(* PLC project Neotec skyrailer, Hydac System GmbH CoDeSys CoDeSys V3.x *)
(* stored: companyURL http://www.hydac.com/, contentDescription This content was automatically generated. Please do not edit., creationDateTime 2025-04-18T16:40:50.760, modificationDateTime 2025-04-18T16:40:50.760 *)

TYPE EBRAKETESTSELECTED : (GE_OSCI_SERVICE_BRAKE := 0, GE_FIXE_SERVICE_BRAKE := 1, GE_OSCI_PARKING_BRAKE := 2, GE_FIXE_PARKING_BRAKE := 3, GE_SERVICE_BRAKES := 4, GE_PARKING_BRAKES := 5, GE_NO_BRAKE := 6, GE_FIXE_2ND_PARKING_BRAKE := 7, GE_OSCI_2ND_PARKING_BRAKE := 8);
END_TYPE

TYPE ECONTROLPOST : (GE_POST_NO_POST := 0, GE_POST_RADIO := 1, GE_POST_NACELLE := 2, GE_POST_TURRET := 3);
END_TYPE

TYPE ECOUNTRY : (GE_FRANCE := 0, GE_SWITZERLAND := 1, GE_UNITED_KINGDOM := 2, GE_AUSTRALIA := 3);
END_TYPE

TYPE EDIGSTATUS : (GE_DIG_OFF := 0, GE_DIG_ON := 1, GE_DIG_ERROR := 2, GE_DIG_UNDEF := 3);
END_TYPE

TYPE EDISTATE : (GE_DI_OFF := 0, GE_DI_ON := 1, GE_DI_ERROR := 2, GE_DI_UNDEF := 3);
END_TYPE

TYPE EERRORSTATUS48XS : (GE_IO_E_OK := 0, GE_IO_E_BUSY := 2, GE_IO_E_UNKNOWN := 3, GE_IO_E_CHANNEL_BUSY := 32, GE_IO_E_CHANNEL_NOT_CONFIGURED := 33, GE_IO_E_FET_PROTECTION := 35, GE_IO_E_ADC_NOT_FINISH := 90, GE_IO_E_PWD_CAPTURE_ERROR := 100, GE_IO_E_PWD_NOT_FINISHED := 101, GE_IO_E_PWD_OPEN_LOAD := 102, GE_IO_E_PWD_SHORT_CIRCUIT := 103, GE_IO_E_PWD_TIMER_OVERFLOW := 104, GE_IO_E_PWD_HIGH_LEVEL := 105, GE_IO_E_PWD_LOW_LEVEL := 106, GE_IO_E_PWD_CURRENT_THRESHOLD_HIGH := 107, GE_IO_E_PWD_CURRENT_THRESHOLD_LOW := 108, GE_IO_E_DO_OPEN_LOAD := 110, GE_IO_E_DO_SHORT_CIRCUIT := 111, GE_IO_E_DO_DIAG_NOT_FINISHED := 112);
END_TYPE

TYPE EMANIPULATORPOSITION : (GE_NEUTRAL := 0, GE_AV := 1, GE_AR := 2, GE_ERROR := 3);
END_TYPE

TYPE EMOTORSTATE : (GE_Stopped := 0, GE_PreStart := 1, GE_Starting := 2, GE_WarmUp := 3, GE_Running := 4, GE_CoolDown := 5, GE_Stopping := 6, GE_PostRun := 7);
END_TYPE

TYPE EMOVENACELLEMODE : (GE_NO_MODE := 0, GE_OFFRAIL_RADIOCONTOL_MODE := 1, GE_RAIL_NACELLE_MODE := 2, GE_TURRET_MODE := 3);
END_TYPE

TYPE EOFFRAILMODE : (GE_NO_OFFRAIL_MODE := 0, GE_TRANSPORT_OFFRAIL_MODE := 1, GE_WORK_OFFRAIL_MODE := 2, GE_WORSHOP_OFFRAIL_MODE := 3);
END_TYPE

TYPE EPOSJOY : (GE_AV_JOY := 0, GE_NEU_JOY := 1, GE_AR_JOY := 2);
END_TYPE

TYPE EPROSTATUS : (GE_PRO_OFF := 0, GE_PRO_ON := 1, GE_PRO_ERROR := 2, GE_PRO_NOT_INSTALLED := 3, GE_PRO_NO_DUTY_CYCLE := 4, GE_PRO_MIN_DUTY_CYCLE := 5);
END_TYPE

TYPE ERAILSPEEDMODE : (GE_NO_SPEED_MAX_RAIL_MODE := 0, GE_ACCESS_SITE_MODE := 1, GE_HIGH_SPEED := 2, GE_LOW_SPEED := 3, GE_LOW_SPEED_BRAKE_TEST_NEEDED := 4, GE_BRAKE_TEST_SPEED_RUNNING := 5, GE_BREAK_IN_BRAKE_SPEED_RUNNING := 6);
END_TYPE

TYPE ERAILTRANSLATIONDIRECTION : (GE_AV_RAIL_DIR := 0, GE_AR_RAIL_DIR := 1, GE_STOP_RAIL_DIR := 2);
END_TYPE

TYPE ERAILWORKMODE : (GE_NO_RAIL_WORK_MODE := 0, GE_BILATERAL_MODE := 1, GE_ALO_MODE := 2, GE_MULTILANE_MODE := 3);
END_TYPE

TYPE ESTATEBOOL2BITS : (GE_OFF := 0, GE_ON := 1, GE_ERR := 2, GE_NA := 3);
END_TYPE

TYPE ESTATEHEARTBEAT : (GE_BOOT_UP := 0, GE_STOPPED := 4, GE_OPERATIONAL := 5, GE_PRE_OPERATIONAL := 127);
END_TYPE

TYPE ESTATESERVICEBRAKERAIL : (GE_DEFINE_BRAKE := 0, GE_AV_SERVICE_BRAKE := 1, GE_AR_SERVICE_BRAKE := 2);
END_TYPE

TYPE ETRANSPORTPOSITION : (GE_NO_TRANSPORT_POSITION := 0, GE_OFFRAIL_TRANSPORT_POSITION := 1, GE_RAIL_TRANSPORT_POSITION := 2);
END_TYPE

TYPE EWDSTATE : (GE_RUNNING := 6, GE_TRIGGERED := 9);
END_TYPE

VAR_GLOBAL CONSTANT  (* GlobalConsts *)
  J1939_SA_DISPLAY : BYTE := 16#2f;  (* Display *)
END_VAR

VAR_GLOBAL  (* GCanMessages *)
  g_CanMessages_Msg8C1SendToOpus : Msg8C1SendToOpusMessageClass;
  g_CanMessages_Msg9C1SendToOpus : Msg9C1SendToOpusMessageClass;
  g_CanMessages_Msg1C0SendToEvision7 : Msg1C0SendToEvision7MessageClass;
  g_CanMessages_Msg2C0SendToEvision7 : Msg2C0SendToEvision7MessageClass;
  g_CanMessages_Msg3C0SendToEvision7 : Msg3C0SendToEvision7MessageClass;
  g_CanMessages_Msg4C0SendToEvision7 : Msg4C0SendToEvision7MessageClass;
  g_CanMessages_Msg5C0SendToEvision7 : Msg5C0SendToEvision7MessageClass;
  g_CanMessages_Msg6C0SendToEvision7 : Msg6C0SendToEvision7MessageClass;
  g_CanMessages_Msg7C0SendToEvision7 : Msg7C0SendToEvision7MessageClass;
  g_CanMessages_Msg8C0SendToEvision7 : Msg8C0SendToEvision7MessageClass;
  g_CanMessages_Msg9C0SendToEvision7 : Msg9C0SendToEvision7MessageClass;
  g_CanMessages_Msg10C0SendToEvision7 : Msg10C0SendToEvision7MessageClass;
  g_CanMessages_Msg11C0SendToEvision7 : Msg11C0SendToEvision7MessageClass;
  g_CanMessages_Msg12C0SendToEvision7 : Msg12C0SendToEvision7MessageClass;
  g_CanMessages_Msg13C0SendToEvision7 : Msg13C0SendToEvision7MessageClass;
  g_CanMessages_Msg14C0SendToEvision7 : Msg14C0SendToEvision7MessageClass;
  g_CanMessages_Msg15C0SendToEvision7 : Msg15C0SendToEvision7MessageClass;
  g_CanMessages_MsgDebugC0SendToEvision7 : MsgDebugC0SendToEvision7MessageClass;
  g_CanMessages_Msg1C1SendToEvision7 : Msg1C1SendToEvision7MessageClass;
  g_CanMessages_Msg2C1SendToEvision7 : Msg2C1SendToEvision7MessageClass;
  g_CanMessages_Msg3C1SendToEvision7 : Msg3C1SendToEvision7MessageClass;
  g_CanMessages_Msg4C1SendToEvision7 : Msg4C1SendToEvision7MessageClass;
  g_CanMessages_Msg5C1SendToEvision7 : Msg5C1SendToEvision7MessageClass;
  g_CanMessages_Msg6C1SendToEvision7 : Msg6C1SendToEvision7MessageClass;
  g_CanMessages_Msg7C1SendToEvision7 : Msg7C1SendToEvision7MessageClass;
  g_CanMessages_Msg8C1SendToEvision7 : Msg8C1SendToEvision7MessageClass;
  g_CanMessages_Msg9C1SendToEvision7 : Msg9C1SendToEvision7MessageClass;
  g_CanMessages_Msg10C1SendToEvision7 : Msg10C1SendToEvision7MessageClass;
  g_CanMessages_Msg11C1SendToEvision7 : Msg11C1SendToEvision7MessageClass;
  g_CanMessages_Msg12C1SendToEvision7 : Msg12C1SendToEvision7MessageClass;
  g_CanMessages_Msg13C1SendToEvision7 : Msg13C1SendToEvision7MessageClass;
  g_CanMessages_Msg14C1SendToEvision7 : Msg14C1SendToEvision7MessageClass;
  g_CanMessages_MsgDebugC1SendToEvision7 : MsgDebugC1SendToEvision7MessageClass;
  g_CanMessages_Msg1RcvFromEvision7 : Msg1RcvFromEvision7MessageClass;
END_VAR

VAR_GLOBAL CONSTANT  (* GeneratedCanConsts *)
  CID_MSG8C1SENDTOOPUS : DWORD := 16#506;
  CID_MSG9C1SENDTOOPUS : DWORD := 16#606;
  CID_MSG1C0SENDTOEVISION7 : DWORD := 16#C0D701;
  CID_MSG2C0SENDTOEVISION7 : DWORD := 16#C0D702;
  CID_MSG3C0SENDTOEVISION7 : DWORD := 16#C0D703;
  CID_MSG4C0SENDTOEVISION7 : DWORD := 16#C0D704;
  CID_MSG5C0SENDTOEVISION7 : DWORD := 16#C0D705;
  CID_MSG6C0SENDTOEVISION7 : DWORD := 16#C0D706;
  CID_MSG7C0SENDTOEVISION7 : DWORD := 16#C0D707;
  CID_MSG8C0SENDTOEVISION7 : DWORD := 16#C0D708;
  CID_MSG9C0SENDTOEVISION7 : DWORD := 16#C0D709;
  CID_MSG10C0SENDTOEVISION7 : DWORD := 16#C0D70A;
  CID_MSG11C0SENDTOEVISION7 : DWORD := 16#C0D70B;
  CID_MSG12C0SENDTOEVISION7 : DWORD := 16#C0D70C;
  CID_MSG13C0SENDTOEVISION7 : DWORD := 16#C0D70D;
  CID_MSG14C0SENDTOEVISION7 : DWORD := 16#C0D70E;
  CID_MSG15C0SENDTOEVISION7 : DWORD := 16#C0D70F;
  CID_MSGDEBUGC0SENDTOEVISION7 : DWORD := 16#C0D711;
  CID_MSG1C1SENDTOEVISION7 : DWORD := 16#C1D701;
  CID_MSG2C1SENDTOEVISION7 : DWORD := 16#C1D702;
  CID_MSG3C1SENDTOEVISION7 : DWORD := 16#C1D703;
  CID_MSG4C1SENDTOEVISION7 : DWORD := 16#C1D704;
  CID_MSG5C1SENDTOEVISION7 : DWORD := 16#C1D705;
  CID_MSG6C1SENDTOEVISION7 : DWORD := 16#C1D706;
  CID_MSG7C1SENDTOEVISION7 : DWORD := 16#C1D707;
  CID_MSG8C1SENDTOEVISION7 : DWORD := 16#C1D708;
  CID_MSG9C1SENDTOEVISION7 : DWORD := 16#C1D709;
  CID_MSG10C1SENDTOEVISION7 : DWORD := 16#C1D70A;
  CID_MSG11C1SENDTOEVISION7 : DWORD := 16#C1D70B;
  CID_MSG12C1SENDTOEVISION7 : DWORD := 16#C1D70C;
  CID_MSG13C1SENDTOEVISION7 : DWORD := 16#C1D70D;
  CID_MSG14C1SENDTOEVISION7 : DWORD := 16#C1D70E;
  CID_MSGDEBUGC1SENDTOEVISION7 : DWORD := 16#C1D712;
  CID_MSG1RCVFROMEVISION7 : DWORD := 16#D7CF01;
END_VAR

VAR_GLOBAL CONSTANT  (* GConsts *)
  J1939_SA_C0 : BYTE := 16#20;
  J1939_SA_C1 : BYTE := 16#21;
  J1939_SA_C2 : BYTE := 16#2F;
  CID_P2P_C0 : DWORD := 16#18EE0020;
  CID_P2P_C1 : DWORD := 16#18EE0021;
END_VAR

FUNCTION_BLOCK CanDispatcherClass IMPLEMENTS ICanDispatcher
  VAR
    fMessage : VBasic.CanMessageClass;
    cycleTimerHst : IntervalTimerClass;  (* Determines how much time lays between the sending of HST can messages (CAN 0) *)
    can0 : VBasic.CanManagerClass;  (* CAN 0: C0_C1_CAN_0 *)
    j1939_can0 : J1939ReceiverClass;
    can1 : VBasic.CanManagerClass;  (* CAN 1: CO_C1_CAN_1_TTC48XS *)
    j1939_can1 : J1939ReceiverClass;
  END_VAR
  VAR_INPUT
    Can0MessagesSent : BoolCanSignalClass;
    Can1MessagesSent : BoolCanSignalClass;
  END_VAR

            
          

METHOD Initialize
                  // **********************************************************************************************************************
// *  AUTO-GENERATED:  PdtCodeBuilder.dll (Version: 1.2.7, Build: 080)
// *  Itf-Version:     1.7.0
// *  Pdt-Version:     2.11.72.172
// *  Pdt-ProjVersion: 0.0.0
// *  Match-Version:   07.04.00.00
// *  Copyright (C) 2012 HYDAC SYSTEM GMBH -  All rights reserved.
// *  Entwicklungsbüro Berlin - Zum Kiesberg 16 - D-14979 Großbeeren
// *  2025-04-18 16:40:50 created
// **********************************************************************************************************************

// Initialize the can bus objects

can0.NetId := 0;
can0.Baudrate := eCanBaudrate.BAUDRATE_250_KBITS;
can0.Initialize();

g_CanMessages_Msg1C0SendToEvision7.Initialize(ADR(can0), CID_MSG1C0SENDTOEVISION7, TCanMessageType.RX, 1000(*Timeout*), 0(*Spn*), 255(*Fmi*), 255(*FmiExt*), eErrorType.ERROR(*ErrType*), eErrorSeverity.CAT0_NO(*ErrCat*), eCanIdFormat.EXTENDED);
g_CanMessages_Msg2C0SendToEvision7.Initialize(ADR(can0), CID_MSG2C0SENDTOEVISION7, TCanMessageType.RX, 1000(*Timeout*), 0(*Spn*), 255(*Fmi*), 255(*FmiExt*), eErrorType.ERROR(*ErrType*), eErrorSeverity.CAT0_NO(*ErrCat*), eCanIdFormat.EXTENDED);
g_CanMessages_Msg3C0SendToEvision7.Initialize(ADR(can0), CID_MSG3C0SENDTOEVISION7, TCanMessageType.RX, 1000(*Timeout*), 0(*Spn*), 255(*Fmi*), 255(*FmiExt*), eErrorType.ERROR(*ErrType*), eErrorSeverity.CAT0_NO(*ErrCat*), eCanIdFormat.EXTENDED);
g_CanMessages_Msg4C0SendToEvision7.Initialize(ADR(can0), CID_MSG4C0SENDTOEVISION7, TCanMessageType.RX, 1000(*Timeout*), 0(*Spn*), 255(*Fmi*), 255(*FmiExt*), eErrorType.ERROR(*ErrType*), eErrorSeverity.CAT0_NO(*ErrCat*), eCanIdFormat.EXTENDED);
g_CanMessages_Msg5C0SendToEvision7.Initialize(ADR(can0), CID_MSG5C0SENDTOEVISION7, TCanMessageType.RX, 1000(*Timeout*), 0(*Spn*), 255(*Fmi*), 255(*FmiExt*), eErrorType.ERROR(*ErrType*), eErrorSeverity.CAT0_NO(*ErrCat*), eCanIdFormat.EXTENDED);
g_CanMessages_Msg6C0SendToEvision7.Initialize(ADR(can0), CID_MSG6C0SENDTOEVISION7, TCanMessageType.RX, 1000(*Timeout*), 0(*Spn*), 255(*Fmi*), 255(*FmiExt*), eErrorType.ERROR(*ErrType*), eErrorSeverity.CAT0_NO(*ErrCat*), eCanIdFormat.EXTENDED);
g_CanMessages_Msg7C0SendToEvision7.Initialize(ADR(can0), CID_MSG7C0SENDTOEVISION7, TCanMessageType.RX, 1000(*Timeout*), 0(*Spn*), 255(*Fmi*), 255(*FmiExt*), eErrorType.ERROR(*ErrType*), eErrorSeverity.CAT0_NO(*ErrCat*), eCanIdFormat.EXTENDED);
g_CanMessages_Msg8C0SendToEvision7.Initialize(ADR(can0), CID_MSG8C0SENDTOEVISION7, TCanMessageType.RX, 1000(*Timeout*), 0(*Spn*), 255(*Fmi*), 255(*FmiExt*), eErrorType.ERROR(*ErrType*), eErrorSeverity.CAT0_NO(*ErrCat*), eCanIdFormat.EXTENDED);
g_CanMessages_Msg9C0SendToEvision7.Initialize(ADR(can0), CID_MSG9C0SENDTOEVISION7, TCanMessageType.RX, 1000(*Timeout*), 0(*Spn*), 255(*Fmi*), 255(*FmiExt*), eErrorType.ERROR(*ErrType*), eErrorSeverity.CAT0_NO(*ErrCat*), eCanIdFormat.EXTENDED);
g_CanMessages_Msg10C0SendToEvision7.Initialize(ADR(can0), CID_MSG10C0SENDTOEVISION7, TCanMessageType.RX, 1000(*Timeout*), 0(*Spn*), 255(*Fmi*), 255(*FmiExt*), eErrorType.ERROR(*ErrType*), eErrorSeverity.CAT0_NO(*ErrCat*), eCanIdFormat.EXTENDED);
g_CanMessages_Msg11C0SendToEvision7.Initialize(ADR(can0), CID_MSG11C0SENDTOEVISION7, TCanMessageType.RX, 1000(*Timeout*), 0(*Spn*), 255(*Fmi*), 255(*FmiExt*), eErrorType.ERROR(*ErrType*), eErrorSeverity.CAT0_NO(*ErrCat*), eCanIdFormat.EXTENDED);
g_CanMessages_Msg12C0SendToEvision7.Initialize(ADR(can0), CID_MSG12C0SENDTOEVISION7, TCanMessageType.RX, 1000(*Timeout*), 0(*Spn*), 255(*Fmi*), 255(*FmiExt*), eErrorType.ERROR(*ErrType*), eErrorSeverity.CAT0_NO(*ErrCat*), eCanIdFormat.EXTENDED);
g_CanMessages_Msg13C0SendToEvision7.Initialize(ADR(can0), CID_MSG13C0SENDTOEVISION7, TCanMessageType.RX, 1000(*Timeout*), 0(*Spn*), 255(*Fmi*), 255(*FmiExt*), eErrorType.ERROR(*ErrType*), eErrorSeverity.CAT0_NO(*ErrCat*), eCanIdFormat.EXTENDED);
g_CanMessages_Msg14C0SendToEvision7.Initialize(ADR(can0), CID_MSG14C0SENDTOEVISION7, TCanMessageType.RX, 1000(*Timeout*), 1544(*Spn*), 31(*Fmi*), 255(*FmiExt*), eErrorType.ERROR(*ErrType*), eErrorSeverity.CAT0_NO(*ErrCat*), eCanIdFormat.EXTENDED);
g_CanMessages_Msg15C0SendToEvision7.Initialize(ADR(can0), CID_MSG15C0SENDTOEVISION7, TCanMessageType.RX, 1000(*Timeout*), 1555(*Spn*), 31(*Fmi*), 255(*FmiExt*), eErrorType.ERROR(*ErrType*), eErrorSeverity.CAT0_NO(*ErrCat*), eCanIdFormat.EXTENDED);
g_CanMessages_MsgDebugC0SendToEvision7.Initialize(ADR(can0), CID_MSGDEBUGC0SENDTOEVISION7, TCanMessageType.RX, 1000(*Timeout*), 0(*Spn*), 255(*Fmi*), 255(*FmiExt*), eErrorType.ERROR(*ErrType*), eErrorSeverity.CAT0_NO(*ErrCat*), eCanIdFormat.EXTENDED);
g_CanMessages_Msg1C1SendToEvision7.Initialize(ADR(can0), CID_MSG1C1SENDTOEVISION7, TCanMessageType.RX, 1000(*Timeout*), 0(*Spn*), 255(*Fmi*), 255(*FmiExt*), eErrorType.ERROR(*ErrType*), eErrorSeverity.CAT0_NO(*ErrCat*), eCanIdFormat.EXTENDED);
g_CanMessages_Msg2C1SendToEvision7.Initialize(ADR(can0), CID_MSG2C1SENDTOEVISION7, TCanMessageType.RX, 1000(*Timeout*), 0(*Spn*), 255(*Fmi*), 255(*FmiExt*), eErrorType.ERROR(*ErrType*), eErrorSeverity.CAT0_NO(*ErrCat*), eCanIdFormat.EXTENDED);
g_CanMessages_Msg3C1SendToEvision7.Initialize(ADR(can0), CID_MSG3C1SENDTOEVISION7, TCanMessageType.RX, 1000(*Timeout*), 0(*Spn*), 255(*Fmi*), 255(*FmiExt*), eErrorType.ERROR(*ErrType*), eErrorSeverity.CAT0_NO(*ErrCat*), eCanIdFormat.EXTENDED);
g_CanMessages_Msg4C1SendToEvision7.Initialize(ADR(can0), CID_MSG4C1SENDTOEVISION7, TCanMessageType.RX, 1000(*Timeout*), 0(*Spn*), 255(*Fmi*), 255(*FmiExt*), eErrorType.ERROR(*ErrType*), eErrorSeverity.CAT0_NO(*ErrCat*), eCanIdFormat.EXTENDED);
g_CanMessages_Msg5C1SendToEvision7.Initialize(ADR(can0), CID_MSG5C1SENDTOEVISION7, TCanMessageType.RX, 1000(*Timeout*), 0(*Spn*), 255(*Fmi*), 255(*FmiExt*), eErrorType.ERROR(*ErrType*), eErrorSeverity.CAT0_NO(*ErrCat*), eCanIdFormat.EXTENDED);
g_CanMessages_Msg6C1SendToEvision7.Initialize(ADR(can0), CID_MSG6C1SENDTOEVISION7, TCanMessageType.RX, 1000(*Timeout*), 0(*Spn*), 255(*Fmi*), 255(*FmiExt*), eErrorType.ERROR(*ErrType*), eErrorSeverity.CAT0_NO(*ErrCat*), eCanIdFormat.EXTENDED);
g_CanMessages_Msg7C1SendToEvision7.Initialize(ADR(can0), CID_MSG7C1SENDTOEVISION7, TCanMessageType.RX, 1000(*Timeout*), 0(*Spn*), 255(*Fmi*), 255(*FmiExt*), eErrorType.ERROR(*ErrType*), eErrorSeverity.CAT0_NO(*ErrCat*), eCanIdFormat.EXTENDED);
g_CanMessages_Msg8C1SendToEvision7.Initialize(ADR(can0), CID_MSG8C1SENDTOEVISION7, TCanMessageType.RX, 1000(*Timeout*), 0(*Spn*), 255(*Fmi*), 255(*FmiExt*), eErrorType.ERROR(*ErrType*), eErrorSeverity.CAT0_NO(*ErrCat*), eCanIdFormat.EXTENDED);
g_CanMessages_Msg9C1SendToEvision7.Initialize(ADR(can0), CID_MSG9C1SENDTOEVISION7, TCanMessageType.RX, 1000(*Timeout*), 0(*Spn*), 255(*Fmi*), 255(*FmiExt*), eErrorType.ERROR(*ErrType*), eErrorSeverity.CAT0_NO(*ErrCat*), eCanIdFormat.EXTENDED);
g_CanMessages_Msg10C1SendToEvision7.Initialize(ADR(can0), CID_MSG10C1SENDTOEVISION7, TCanMessageType.RX, 1000(*Timeout*), 0(*Spn*), 255(*Fmi*), 255(*FmiExt*), eErrorType.ERROR(*ErrType*), eErrorSeverity.CAT0_NO(*ErrCat*), eCanIdFormat.EXTENDED);
g_CanMessages_Msg11C1SendToEvision7.Initialize(ADR(can0), CID_MSG11C1SENDTOEVISION7, TCanMessageType.RX, 1000(*Timeout*), 0(*Spn*), 255(*Fmi*), 255(*FmiExt*), eErrorType.ERROR(*ErrType*), eErrorSeverity.CAT0_NO(*ErrCat*), eCanIdFormat.EXTENDED);
g_CanMessages_Msg12C1SendToEvision7.Initialize(ADR(can0), CID_MSG12C1SENDTOEVISION7, TCanMessageType.RX, 1000(*Timeout*), 0(*Spn*), 255(*Fmi*), 255(*FmiExt*), eErrorType.ERROR(*ErrType*), eErrorSeverity.CAT0_NO(*ErrCat*), eCanIdFormat.EXTENDED);
g_CanMessages_Msg13C1SendToEvision7.Initialize(ADR(can0), CID_MSG13C1SENDTOEVISION7, TCanMessageType.RX, 1000(*Timeout*), 0(*Spn*), 255(*Fmi*), 255(*FmiExt*), eErrorType.ERROR(*ErrType*), eErrorSeverity.CAT0_NO(*ErrCat*), eCanIdFormat.EXTENDED);
g_CanMessages_Msg14C1SendToEvision7.Initialize(ADR(can0), CID_MSG14C1SENDTOEVISION7, TCanMessageType.RX, 1000(*Timeout*), 1561(*Spn*), 31(*Fmi*), 255(*FmiExt*), eErrorType.ERROR(*ErrType*), eErrorSeverity.CAT0_NO(*ErrCat*), eCanIdFormat.EXTENDED);
g_CanMessages_MsgDebugC1SendToEvision7.Initialize(ADR(can0), CID_MSGDEBUGC1SENDTOEVISION7, TCanMessageType.RX, 1000(*Timeout*), 0(*Spn*), 255(*Fmi*), 255(*FmiExt*), eErrorType.ERROR(*ErrType*), eErrorSeverity.CAT0_NO(*ErrCat*), eCanIdFormat.EXTENDED);
g_CanMessages_Msg1RcvFromEvision7.Initialize(ADR(can0), CID_MSG1RCVFROMEVISION7, TCanMessageType.TXC, 20(*CycleTime*), 10(*MinimumCycleTime*), 50(*StartOffset*), eCanIdFormat.EXTENDED);

can1.NetId := 1;
can1.Baudrate := eCanBaudrate.BAUDRATE_500_KBITS;
can1.Initialize();

g_CanMessages_Msg8C1SendToOpus.Initialize(ADR(can1), CID_MSG8C1SENDTOOPUS, TCanMessageType.RX, 1000(*Timeout*), 0(*Spn*), 255(*Fmi*), 255(*FmiExt*), eErrorType.ERROR(*ErrType*), eErrorSeverity.CAT0_NO(*ErrCat*), eCanIdFormat.STANDARD);
g_CanMessages_Msg9C1SendToOpus.Initialize(ADR(can1), CID_MSG9C1SENDTOOPUS, TCanMessageType.RX, 1000(*Timeout*), 1537(*Spn*), 31(*Fmi*), 255(*FmiExt*), eErrorType.ERROR(*ErrType*), eErrorSeverity.CAT0_NO(*ErrCat*), eCanIdFormat.STANDARD);

// Initialize J1939:
j1939_can0.Initialize(ADR(can0.ReceiverManager));
j1939_can1.Initialize(ADR(can1.ReceiverManager));

// DM1 on CAN-Bus 0:
gLib_Dm1ErrorListManager.AddDm1SourceAddress(ADR(j1939_can0), J1939_SA_C0, DtcVersion.DtcVersion1);
// DM1 on CAN-Bus 0:
gLib_Dm1ErrorListManager.AddDm1SourceAddress(ADR(j1939_can0), J1939_SA_C1, DtcVersion.DtcVersion1);

                
END_METHOD

METHOD InvalidateRead
                  _processCan0Read();
_processCan1Read();

_processJ1939();


                
END_METHOD

METHOD InvalidateWrite
                  _processCan0Write();
_processCan1Write();


                
END_METHOD

METHOD _processCan0Read
  VAR
    canMsg : CanMessageClass;
    messageCount : INT;
    synConnection : BOOL;
  END_VAR
                  canMsg := Can0.ReceivedMessage;
WHILE canMsg.NewData DO
	CASE canMsg.CobId OF
		CID_MSG1C0SENDTOEVISION7:
			g_CanMessages_Msg1C0SendToEvision7.SetData(ADR(canMsg));
		CID_MSG2C0SENDTOEVISION7:
			g_CanMessages_Msg2C0SendToEvision7.SetData(ADR(canMsg));
		CID_MSG3C0SENDTOEVISION7:
			g_CanMessages_Msg3C0SendToEvision7.SetData(ADR(canMsg));
		CID_MSG4C0SENDTOEVISION7:
			g_CanMessages_Msg4C0SendToEvision7.SetData(ADR(canMsg));
		CID_MSG5C0SENDTOEVISION7:
			g_CanMessages_Msg5C0SendToEvision7.SetData(ADR(canMsg));
		CID_MSG6C0SENDTOEVISION7:
			g_CanMessages_Msg6C0SendToEvision7.SetData(ADR(canMsg));
		CID_MSG7C0SENDTOEVISION7:
			g_CanMessages_Msg7C0SendToEvision7.SetData(ADR(canMsg));
		CID_MSG8C0SENDTOEVISION7:
			g_CanMessages_Msg8C0SendToEvision7.SetData(ADR(canMsg));
		CID_MSG9C0SENDTOEVISION7:
			g_CanMessages_Msg9C0SendToEvision7.SetData(ADR(canMsg));
		CID_MSG10C0SENDTOEVISION7:
			g_CanMessages_Msg10C0SendToEvision7.SetData(ADR(canMsg));
		CID_MSG11C0SENDTOEVISION7:
			g_CanMessages_Msg11C0SendToEvision7.SetData(ADR(canMsg));
		CID_MSG12C0SENDTOEVISION7:
			g_CanMessages_Msg12C0SendToEvision7.SetData(ADR(canMsg));
		CID_MSG13C0SENDTOEVISION7:
			g_CanMessages_Msg13C0SendToEvision7.SetData(ADR(canMsg));
		CID_MSG14C0SENDTOEVISION7:
			g_CanMessages_Msg14C0SendToEvision7.SetData(ADR(canMsg));
		CID_MSG15C0SENDTOEVISION7:
			g_CanMessages_Msg15C0SendToEvision7.SetData(ADR(canMsg));
		CID_MSGDEBUGC0SENDTOEVISION7:
			g_CanMessages_MsgDebugC0SendToEvision7.SetData(ADR(canMsg));
		CID_MSG1C1SENDTOEVISION7:
			g_CanMessages_Msg1C1SendToEvision7.SetData(ADR(canMsg));
		CID_MSG2C1SENDTOEVISION7:
			g_CanMessages_Msg2C1SendToEvision7.SetData(ADR(canMsg));
		CID_MSG3C1SENDTOEVISION7:
			g_CanMessages_Msg3C1SendToEvision7.SetData(ADR(canMsg));
		CID_MSG4C1SENDTOEVISION7:
			g_CanMessages_Msg4C1SendToEvision7.SetData(ADR(canMsg));
		CID_MSG5C1SENDTOEVISION7:
			g_CanMessages_Msg5C1SendToEvision7.SetData(ADR(canMsg));
		CID_MSG6C1SENDTOEVISION7:
			g_CanMessages_Msg6C1SendToEvision7.SetData(ADR(canMsg));
		CID_MSG7C1SENDTOEVISION7:
			g_CanMessages_Msg7C1SendToEvision7.SetData(ADR(canMsg));
		CID_MSG8C1SENDTOEVISION7:
			g_CanMessages_Msg8C1SendToEvision7.SetData(ADR(canMsg));
		CID_MSG9C1SENDTOEVISION7:
			g_CanMessages_Msg9C1SendToEvision7.SetData(ADR(canMsg));
		CID_MSG10C1SENDTOEVISION7:
			g_CanMessages_Msg10C1SendToEvision7.SetData(ADR(canMsg));
		CID_MSG11C1SENDTOEVISION7:
			g_CanMessages_Msg11C1SendToEvision7.SetData(ADR(canMsg));
		CID_MSG12C1SENDTOEVISION7:
			g_CanMessages_Msg12C1SendToEvision7.SetData(ADR(canMsg));
		CID_MSG13C1SENDTOEVISION7:
			g_CanMessages_Msg13C1SendToEvision7.SetData(ADR(canMsg));
		CID_MSG14C1SENDTOEVISION7:
			g_CanMessages_Msg14C1SendToEvision7.SetData(ADR(canMsg));
		CID_MSGDEBUGC1SENDTOEVISION7:
			g_CanMessages_MsgDebugC1SendToEvision7.SetData(ADR(canMsg));
		CID_P2P_C0,
		CID_P2P_C1:
			;
	ELSE
		IF ( NOT gLib_HstCommunicator.ProcessHstProtocol(ADR(canMsg)) ) THEN
			j1939_can0.ProcessCanMessage(ADR(canMsg));
		END_IF
	END_CASE

	//Message counter
	messageCount := messageCount + 1;
	IF messageCount = 200 THEN
		FastLog(LogClass.LOG_WARNING, 'Message count over 200 CAN0');
		EXIT;
	ELSE
		canMsg := Can0.ReceivedMessage;
	END_IF
END_WHILE

_invalidateCan0ReceiveMessages();

                
END_METHOD

METHOD _invalidateCan0ReceiveMessages
                  g_CanMessages_Msg1C0SendToEvision7.InvalidateNonVisuals();
g_CanMessages_Msg2C0SendToEvision7.InvalidateNonVisuals();
g_CanMessages_Msg3C0SendToEvision7.InvalidateNonVisuals();
g_CanMessages_Msg4C0SendToEvision7.InvalidateNonVisuals();
g_CanMessages_Msg5C0SendToEvision7.InvalidateNonVisuals();
g_CanMessages_Msg6C0SendToEvision7.InvalidateNonVisuals();
g_CanMessages_Msg7C0SendToEvision7.InvalidateNonVisuals();
g_CanMessages_Msg8C0SendToEvision7.InvalidateNonVisuals();
g_CanMessages_Msg9C0SendToEvision7.InvalidateNonVisuals();
g_CanMessages_Msg10C0SendToEvision7.InvalidateNonVisuals();
g_CanMessages_Msg11C0SendToEvision7.InvalidateNonVisuals();
g_CanMessages_Msg12C0SendToEvision7.InvalidateNonVisuals();
g_CanMessages_Msg13C0SendToEvision7.InvalidateNonVisuals();
g_CanMessages_Msg14C0SendToEvision7.InvalidateNonVisuals();
g_CanMessages_Msg15C0SendToEvision7.InvalidateNonVisuals();
g_CanMessages_MsgDebugC0SendToEvision7.InvalidateNonVisuals();
g_CanMessages_Msg1C1SendToEvision7.InvalidateNonVisuals();
g_CanMessages_Msg2C1SendToEvision7.InvalidateNonVisuals();
g_CanMessages_Msg3C1SendToEvision7.InvalidateNonVisuals();
g_CanMessages_Msg4C1SendToEvision7.InvalidateNonVisuals();
g_CanMessages_Msg5C1SendToEvision7.InvalidateNonVisuals();
g_CanMessages_Msg6C1SendToEvision7.InvalidateNonVisuals();
g_CanMessages_Msg7C1SendToEvision7.InvalidateNonVisuals();
g_CanMessages_Msg8C1SendToEvision7.InvalidateNonVisuals();
g_CanMessages_Msg9C1SendToEvision7.InvalidateNonVisuals();
g_CanMessages_Msg10C1SendToEvision7.InvalidateNonVisuals();
g_CanMessages_Msg11C1SendToEvision7.InvalidateNonVisuals();
g_CanMessages_Msg12C1SendToEvision7.InvalidateNonVisuals();
g_CanMessages_Msg13C1SendToEvision7.InvalidateNonVisuals();
g_CanMessages_Msg14C1SendToEvision7.InvalidateNonVisuals();
g_CanMessages_MsgDebugC1SendToEvision7.InvalidateNonVisuals();

                
END_METHOD

METHOD _processJ1939Sub
  VAR_INPUT
    pJ1939Msg : POINTER TO J1939MessageClass;
  END_VAR
                  IF IsValidPointer(pJ1939Msg, 'CanDispatcherClass._processJ1939Sub') AND pJ1939Msg^.IsFinished THEN
	CASE pJ1939Msg^.PGN OF
		J1939_PGN_DM1:
			gLib_Dm1ErrorListManager.ProcessDm1Message(pJ1939Msg);
	END_CASE
END_IF

                
END_METHOD

METHOD _processCan0Write
                  _invalidateCan0TransmitMessages();

IF cycleTimerHst.IntervalReached THEN
	gLib_HstCommunicator.SendHstCommand();
END_IF

                
END_METHOD

METHOD _invalidateCan0TransmitMessages
                  g_CanMessages_Msg1RcvFromEvision7.InvalidateNonVisuals();

                
END_METHOD

PROPERTY CanBus0 : POINTER TO CanManagerClass
GET
                    CanBus0 := ADR(can0);

                  
END_GET
END_PROPERTY

METHOD _processCan1Read
  VAR
    canMsg : CanMessageClass;
    messageCount : INT;
  END_VAR
                  canMsg := Can1.ReceivedMessage;
WHILE canMsg.NewData DO
	CASE canMsg.CobId OF
		CID_MSG8C1SENDTOOPUS:
			g_CanMessages_Msg8C1SendToOpus.SetData(ADR(canMsg));
		CID_MSG9C1SENDTOOPUS:
			g_CanMessages_Msg9C1SendToOpus.SetData(ADR(canMsg));
	ELSE
		j1939_can1.ProcessCanMessage(ADR(canMsg));
	END_CASE

	//Message counter
	messageCount := messageCount + 1;
	IF messageCount = 200 THEN
		FastLog(LogClass.LOG_WARNING, 'Message count over 200 CAN1');
		EXIT;
	ELSE
		canMsg := Can1.ReceivedMessage;
	END_IF
END_WHILE

_invalidateCan1ReceiveMessages();

                
END_METHOD

METHOD _invalidateCan1ReceiveMessages
                  g_CanMessages_Msg8C1SendToOpus.InvalidateNonVisuals();
g_CanMessages_Msg9C1SendToOpus.InvalidateNonVisuals();

                
END_METHOD

METHOD _processCan1Write
                  _invalidateCan1TransmitMessages();

                
END_METHOD

METHOD _invalidateCan1TransmitMessages
                  
                
END_METHOD

PROPERTY CanBus1 : POINTER TO CanManagerClass
GET
                    CanBus1 := ADR(can1);

                  
END_GET
END_PROPERTY

METHOD _processJ1939
  VAR
    j1939Msg : J1939MessageClass;
  END_VAR
                  // Process CAN-0 messages:
j1939Msg := j1939_can0.GetNextNewMessage();
_processJ1939Sub(ADR(j1939Msg));

// Process CAN-1 messages:
j1939Msg := j1939_can1.GetNextNewMessage();
_processJ1939Sub(ADR(j1939Msg));


                
END_METHOD
END_FUNCTION_BLOCK

FUNCTION_BLOCK Msg1C0SendToEvision7MessageClass EXTENDS CanReceiveMessageClass
  VAR_INPUT
    bogBreak_Parking_On_Off : BoolCanSignalClass;
    bogBreak_Faillure_On_Off : BoolCanSignalClass;
    bogMovement_Allow_Nacelle : BoolCanSignalClass;
    bogTurretSectorInCenter : BoolCanSignalClass;
    bogTurretInCenter : BoolCanSignalClass;
    bogVehiculeTrainMode : BoolCanSignalClass;
    bogIncoherenceLateralStopAndKey : BoolCanSignalClass;
    bogWorkMode : BoolCanSignalClass;
    bogSafetyElectricPump : BoolCanSignalClass;
    bogDownhill150mm : BoolCanSignalClass;
    bogTrainModeAllow : BoolCanSignalClass;
    bogBrakeTestService : BoolCanSignalClass;
    bogBrakePressureFault : BoolCanSignalClass;
    bogActivateMeasuringMast : BoolCanSignalClass;
    bogAutoMovementDirectionLight : BoolCanSignalClass;
    bogBackRailwayAxleLowPosition : BoolCanSignalClass;
    bogFrontRailwayAxleLowPosition : BoolCanSignalClass;
    bogBackRailwayAxleServiceBrake : BoolCanSignalClass;
    bogFrontRailwayAxleServiceBrake : BoolCanSignalClass;
    bogBackRailwayAxleParkBrake : BoolCanSignalClass;
    bogFrontRailwayAxleParkBrake : BoolCanSignalClass;
    bogStatusFrontLeftTrainBrakeTest : BoolCanSignalClass;
    bogStatFrontRightTrainBrakeTest : BoolCanSignalClass;
    bogStatusBackLeftTrainBrakeTest : BoolCanSignalClass;
    bogStatusBackRightTrainBrakeTest : BoolCanSignalClass;
    bogAlarmAru : BoolCanSignalClass;
    bogLitmitSpeedExceeded : BoolCanSignalClass;
    bogShowCamera : BoolCanSignalClass;
    bogFixeAxleFrequencyFault : BoolCanSignalClass;
    bogOscillantAxleFrequencyFault : BoolCanSignalClass;
    bogTemperatureTransmAlarm : BoolCanSignalClass;
    bogUserCodeOption : BoolCanSignalClass;
    bogRequestForwardTransRail : BoolCanSignalClass;
    bogRequestBackwardTransRail : BoolCanSignalClass;
    bogEvForwardFault : BoolCanSignalClass;
    bogEvBackwardFault : BoolCanSignalClass;
    bogIncoherenceModeTravail : BoolCanSignalClass;
    bogIncoherenceBasketStopAndKey : BoolCanSignalClass;
    bogCenteredAdvanceJoystick : BoolCanSignalClass;
    bogKlaxon : BoolCanSignalClass;
    bogGachette : BoolCanSignalClass;
    bogStopMoteur : BoolCanSignalClass;
    bogEStop : BoolCanSignalClass;
    bogDeadMan : BoolCanSignalClass;
    bogSignalDangerMode : BoolCanSignalClass;
    bogLimitSpeedLowSpeedBrakeTest : BoolCanSignalClass;
    bogSlopeSensorFault : BoolCanSignalClass;
    bogMastMeasureFault : BoolCanSignalClass;
    i16gEncodeurTurretAngle : Int16CanSignalClass;
    Counter : UInt32CanSignalClass;
  END_VAR

            
          

METHOD SetData
  VAR_INPUT
    CanMsgPointer : POINTER TO CanMessageClass;
  END_VAR
                  IF IsValidPointer(canMsgPointer,'SetData') THEN
	SUPER^.SetData(CanMsgPointer);
	//Set the new data
	bogBreak_Parking_On_Off.Value := canMsgPointer^.GetBoolOnBit(0);
	bogBreak_Faillure_On_Off.Value := canMsgPointer^.GetBoolOnBit(1);
	bogMovement_Allow_Nacelle.Value := canMsgPointer^.GetBoolOnBit(2);
	bogTurretSectorInCenter.Value := canMsgPointer^.GetBoolOnBit(3);
	bogTurretInCenter.Value := canMsgPointer^.GetBoolOnBit(4);
	bogVehiculeTrainMode.Value := canMsgPointer^.GetBoolOnBit(5);
	bogIncoherenceLateralStopAndKey.Value := canMsgPointer^.GetBoolOnBit(6);
	bogWorkMode.Value := canMsgPointer^.GetBoolOnBit(7);
	bogSafetyElectricPump.Value := canMsgPointer^.GetBoolOnBit(8);
	bogDownhill150mm.Value := canMsgPointer^.GetBoolOnBit(9);
	bogTrainModeAllow.Value := canMsgPointer^.GetBoolOnBit(10);
	bogBrakeTestService.Value := canMsgPointer^.GetBoolOnBit(11);
	bogBrakePressureFault.Value := canMsgPointer^.GetBoolOnBit(12);
	bogActivateMeasuringMast.Value := canMsgPointer^.GetBoolOnBit(13);
	bogAutoMovementDirectionLight.Value := canMsgPointer^.GetBoolOnBit(14);
	bogBackRailwayAxleLowPosition.Value := canMsgPointer^.GetBoolOnBit(15);
	bogFrontRailwayAxleLowPosition.Value := canMsgPointer^.GetBoolOnBit(16);
	bogBackRailwayAxleServiceBrake.Value := canMsgPointer^.GetBoolOnBit(17);
	bogFrontRailwayAxleServiceBrake.Value := canMsgPointer^.GetBoolOnBit(18);
	bogBackRailwayAxleParkBrake.Value := canMsgPointer^.GetBoolOnBit(19);
	bogFrontRailwayAxleParkBrake.Value := canMsgPointer^.GetBoolOnBit(20);
	bogStatusFrontLeftTrainBrakeTest.Value := canMsgPointer^.GetBoolOnBit(21);
	bogStatFrontRightTrainBrakeTest.Value := canMsgPointer^.GetBoolOnBit(22);
	bogStatusBackLeftTrainBrakeTest.Value := canMsgPointer^.GetBoolOnBit(23);
	bogStatusBackRightTrainBrakeTest.Value := canMsgPointer^.GetBoolOnBit(24);
	bogAlarmAru.Value := canMsgPointer^.GetBoolOnBit(25);
	bogLitmitSpeedExceeded.Value := canMsgPointer^.GetBoolOnBit(26);
	bogShowCamera.Value := canMsgPointer^.GetBoolOnBit(27);
	bogFixeAxleFrequencyFault.Value := canMsgPointer^.GetBoolOnBit(28);
	bogOscillantAxleFrequencyFault.Value := canMsgPointer^.GetBoolOnBit(29);
	bogTemperatureTransmAlarm.Value := canMsgPointer^.GetBoolOnBit(30);
	bogUserCodeOption.Value := canMsgPointer^.GetBoolOnBit(31);
	bogRequestForwardTransRail.Value := canMsgPointer^.GetBoolOnBit(32);
	bogRequestBackwardTransRail.Value := canMsgPointer^.GetBoolOnBit(33);
	bogEvForwardFault.Value := canMsgPointer^.GetBoolOnBit(34);
	bogEvBackwardFault.Value := canMsgPointer^.GetBoolOnBit(35);
	bogIncoherenceModeTravail.Value := canMsgPointer^.GetBoolOnBit(36);
	bogIncoherenceBasketStopAndKey.Value := canMsgPointer^.GetBoolOnBit(37);
	bogCenteredAdvanceJoystick.Value := canMsgPointer^.GetBoolOnBit(38);
	bogKlaxon.Value := canMsgPointer^.GetBoolOnBit(39);
	bogGachette.Value := canMsgPointer^.GetBoolOnBit(40);
	bogStopMoteur.Value := canMsgPointer^.GetBoolOnBit(41);
	bogEStop.Value := canMsgPointer^.GetBoolOnBit(42);
	bogDeadMan.Value := canMsgPointer^.GetBoolOnBit(43);
	bogSignalDangerMode.Value := canMsgPointer^.GetBoolOnBit(44);
	bogLimitSpeedLowSpeedBrakeTest.Value := canMsgPointer^.GetBoolOnBit(45);
	bogSlopeSensorFault.Value := canMsgPointer^.GetBoolOnBit(46);
	bogMastMeasureFault.Value := canMsgPointer^.GetBoolOnBit(47);
	i16gEncodeurTurretAngle.Value := canMsgPointer^.GetInt16(48);
	//And increase the counter
	Counter.Value := CanMsgPointer^.Counter.Value;
END_IF

                
END_METHOD

PROPERTY bogBreak_Parking_On_OffRawValue : BOOL
GET
                    bogBreak_Parking_On_OffRawValue := bogBreak_Parking_On_Off.Value;

                  
END_GET
END_PROPERTY

PROPERTY bogBreak_Faillure_On_OffRawValue : BOOL
GET
                    bogBreak_Faillure_On_OffRawValue := bogBreak_Faillure_On_Off.Value;

                  
END_GET
END_PROPERTY

PROPERTY bogMovement_Allow_NacelleRawValue : BOOL
GET
                    bogMovement_Allow_NacelleRawValue := bogMovement_Allow_Nacelle.Value;

                  
END_GET
END_PROPERTY

PROPERTY bogTurretSectorInCenterRawValue : BOOL
GET
                    bogTurretSectorInCenterRawValue := bogTurretSectorInCenter.Value;

                  
END_GET
END_PROPERTY

PROPERTY bogTurretInCenterRawValue : BOOL
GET
                    bogTurretInCenterRawValue := bogTurretInCenter.Value;

                  
END_GET
END_PROPERTY

PROPERTY bogVehiculeTrainModeRawValue : BOOL
GET
                    bogVehiculeTrainModeRawValue := bogVehiculeTrainMode.Value;

                  
END_GET
END_PROPERTY

PROPERTY bogIncoherenceLateralStopAndKeyRawValue : BOOL
GET
                    bogIncoherenceLateralStopAndKeyRawValue := bogIncoherenceLateralStopAndKey.Value;

                  
END_GET
END_PROPERTY

PROPERTY bogWorkModeRawValue : BOOL
GET
                    bogWorkModeRawValue := bogWorkMode.Value;

                  
END_GET
END_PROPERTY

PROPERTY bogSafetyElectricPumpRawValue : BOOL
GET
                    bogSafetyElectricPumpRawValue := bogSafetyElectricPump.Value;

                  
END_GET
END_PROPERTY

PROPERTY bogDownhill150mmRawValue : BOOL
GET
                    bogDownhill150mmRawValue := bogDownhill150mm.Value;

                  
END_GET
END_PROPERTY

PROPERTY bogTrainModeAllowRawValue : BOOL
GET
                    bogTrainModeAllowRawValue := bogTrainModeAllow.Value;

                  
END_GET
END_PROPERTY

PROPERTY bogBrakeTestServiceRawValue : BOOL
GET
                    bogBrakeTestServiceRawValue := bogBrakeTestService.Value;

                  
END_GET
END_PROPERTY

PROPERTY bogBrakePressureFaultRawValue : BOOL
GET
                    bogBrakePressureFaultRawValue := bogBrakePressureFault.Value;

                  
END_GET
END_PROPERTY

PROPERTY bogActivateMeasuringMastRawValue : BOOL
GET
                    bogActivateMeasuringMastRawValue := bogActivateMeasuringMast.Value;

                  
END_GET
END_PROPERTY

PROPERTY bogAutoMovementDirectionLightRawValue : BOOL
GET
                    bogAutoMovementDirectionLightRawValue := bogAutoMovementDirectionLight.Value;

                  
END_GET
END_PROPERTY

PROPERTY bogBackRailwayAxleLowPositionRawValue : BOOL
GET
                    bogBackRailwayAxleLowPositionRawValue := bogBackRailwayAxleLowPosition.Value;

                  
END_GET
END_PROPERTY

PROPERTY bogFrontRailwayAxleLowPositionRawValue : BOOL
GET
                    bogFrontRailwayAxleLowPositionRawValue := bogFrontRailwayAxleLowPosition.Value;

                  
END_GET
END_PROPERTY

PROPERTY bogBackRailwayAxleServiceBrakeRawValue : BOOL
GET
                    bogBackRailwayAxleServiceBrakeRawValue := bogBackRailwayAxleServiceBrake.Value;

                  
END_GET
END_PROPERTY

PROPERTY bogFrontRailwayAxleServiceBrakeRawValue : BOOL
GET
                    bogFrontRailwayAxleServiceBrakeRawValue := bogFrontRailwayAxleServiceBrake.Value;

                  
END_GET
END_PROPERTY

PROPERTY bogBackRailwayAxleParkBrakeRawValue : BOOL
GET
                    bogBackRailwayAxleParkBrakeRawValue := bogBackRailwayAxleParkBrake.Value;

                  
END_GET
END_PROPERTY

PROPERTY bogFrontRailwayAxleParkBrakeRawValue : BOOL
GET
                    bogFrontRailwayAxleParkBrakeRawValue := bogFrontRailwayAxleParkBrake.Value;

                  
END_GET
END_PROPERTY

PROPERTY bogStatusFrontLeftTrainBrakeTestRawValue : BOOL
GET
                    bogStatusFrontLeftTrainBrakeTestRawValue := bogStatusFrontLeftTrainBrakeTest.Value;

                  
END_GET
END_PROPERTY

PROPERTY bogStatFrontRightTrainBrakeTestRawValue : BOOL
GET
                    bogStatFrontRightTrainBrakeTestRawValue := bogStatFrontRightTrainBrakeTest.Value;

                  
END_GET
END_PROPERTY

PROPERTY bogStatusBackLeftTrainBrakeTestRawValue : BOOL
GET
                    bogStatusBackLeftTrainBrakeTestRawValue := bogStatusBackLeftTrainBrakeTest.Value;

                  
END_GET
END_PROPERTY

PROPERTY bogStatusBackRightTrainBrakeTestRawValue : BOOL
GET
                    bogStatusBackRightTrainBrakeTestRawValue := bogStatusBackRightTrainBrakeTest.Value;

                  
END_GET
END_PROPERTY

PROPERTY bogAlarmAruRawValue : BOOL
GET
                    bogAlarmAruRawValue := bogAlarmAru.Value;

                  
END_GET
END_PROPERTY

PROPERTY bogLitmitSpeedExceededRawValue : BOOL
GET
                    bogLitmitSpeedExceededRawValue := bogLitmitSpeedExceeded.Value;

                  
END_GET
END_PROPERTY

PROPERTY bogShowCameraRawValue : BOOL
GET
                    bogShowCameraRawValue := bogShowCamera.Value;

                  
END_GET
END_PROPERTY

PROPERTY bogFixeAxleFrequencyFaultRawValue : BOOL
GET
                    bogFixeAxleFrequencyFaultRawValue := bogFixeAxleFrequencyFault.Value;

                  
END_GET
END_PROPERTY

PROPERTY bogOscillantAxleFrequencyFaultRawValue : BOOL
GET
                    bogOscillantAxleFrequencyFaultRawValue := bogOscillantAxleFrequencyFault.Value;

                  
END_GET
END_PROPERTY

PROPERTY bogTemperatureTransmAlarmRawValue : BOOL
GET
                    bogTemperatureTransmAlarmRawValue := bogTemperatureTransmAlarm.Value;

                  
END_GET
END_PROPERTY

PROPERTY bogUserCodeOptionRawValue : BOOL
GET
                    bogUserCodeOptionRawValue := bogUserCodeOption.Value;

                  
END_GET
END_PROPERTY

PROPERTY bogRequestForwardTransRailRawValue : BOOL
GET
                    bogRequestForwardTransRailRawValue := bogRequestForwardTransRail.Value;

                  
END_GET
END_PROPERTY

PROPERTY bogRequestBackwardTransRailRawValue : BOOL
GET
                    bogRequestBackwardTransRailRawValue := bogRequestBackwardTransRail.Value;

                  
END_GET
END_PROPERTY

PROPERTY bogEvForwardFaultRawValue : BOOL
GET
                    bogEvForwardFaultRawValue := bogEvForwardFault.Value;

                  
END_GET
END_PROPERTY

PROPERTY bogEvBackwardFaultRawValue : BOOL
GET
                    bogEvBackwardFaultRawValue := bogEvBackwardFault.Value;

                  
END_GET
END_PROPERTY

PROPERTY bogIncoherenceModeTravailRawValue : BOOL
GET
                    bogIncoherenceModeTravailRawValue := bogIncoherenceModeTravail.Value;

                  
END_GET
END_PROPERTY

PROPERTY bogIncoherenceBasketStopAndKeyRawValue : BOOL
GET
                    bogIncoherenceBasketStopAndKeyRawValue := bogIncoherenceBasketStopAndKey.Value;

                  
END_GET
END_PROPERTY

PROPERTY bogCenteredAdvanceJoystickRawValue : BOOL
GET
                    bogCenteredAdvanceJoystickRawValue := bogCenteredAdvanceJoystick.Value;

                  
END_GET
END_PROPERTY

PROPERTY bogKlaxonRawValue : BOOL
GET
                    bogKlaxonRawValue := bogKlaxon.Value;

                  
END_GET
END_PROPERTY

PROPERTY bogGachetteRawValue : BOOL
GET
                    bogGachetteRawValue := bogGachette.Value;

                  
END_GET
END_PROPERTY

PROPERTY bogStopMoteurRawValue : BOOL
GET
                    bogStopMoteurRawValue := bogStopMoteur.Value;

                  
END_GET
END_PROPERTY

PROPERTY bogEStopRawValue : BOOL
GET
                    bogEStopRawValue := bogEStop.Value;

                  
END_GET
END_PROPERTY

PROPERTY bogDeadManRawValue : BOOL
GET
                    bogDeadManRawValue := bogDeadMan.Value;

                  
END_GET
END_PROPERTY

PROPERTY bogSignalDangerModeRawValue : BOOL
GET
                    bogSignalDangerModeRawValue := bogSignalDangerMode.Value;

                  
END_GET
END_PROPERTY

PROPERTY bogLimitSpeedLowSpeedBrakeTestRawValue : BOOL
GET
                    bogLimitSpeedLowSpeedBrakeTestRawValue := bogLimitSpeedLowSpeedBrakeTest.Value;

                  
END_GET
END_PROPERTY

PROPERTY bogSlopeSensorFaultRawValue : BOOL
GET
                    bogSlopeSensorFaultRawValue := bogSlopeSensorFault.Value;

                  
END_GET
END_PROPERTY

PROPERTY bogMastMeasureFaultRawValue : BOOL
GET
                    bogMastMeasureFaultRawValue := bogMastMeasureFault.Value;

                  
END_GET
END_PROPERTY

PROPERTY i16gEncodeurTurretAngleRawValue : INT
GET
                    IF i16gEncodeurTurretAngle.AppScalingMultiplier = 0 THEN
	_MatchLog^.Error("Get i16gEncodeurTurretAngleRawValue", "Division by Zero!");
	RETURN;
End_IF

i16gEncodeurTurretAngleRawValue := TO_INT((i16gEncodeurTurretAngle.Value - i16gEncodeurTurretAngle.AppScalingOffset) * i16gEncodeurTurretAngle.AppScalingDivisor / i16gEncodeurTurretAngle.AppScalingMultiplier);

                  
END_GET
END_PROPERTY

PROPERTY bogBreak_Parking_On_OffToolValue : BOOL
GET
                    bogBreak_Parking_On_OffToolValue := bogBreak_Parking_On_Off.Value;

                  
END_GET
END_PROPERTY

PROPERTY bogBreak_Faillure_On_OffToolValue : BOOL
GET
                    bogBreak_Faillure_On_OffToolValue := bogBreak_Faillure_On_Off.Value;

                  
END_GET
END_PROPERTY

PROPERTY bogMovement_Allow_NacelleToolValue : BOOL
GET
                    bogMovement_Allow_NacelleToolValue := bogMovement_Allow_Nacelle.Value;

                  
END_GET
END_PROPERTY

PROPERTY bogTurretSectorInCenterToolValue : BOOL
GET
                    bogTurretSectorInCenterToolValue := bogTurretSectorInCenter.Value;

                  
END_GET
END_PROPERTY

PROPERTY bogTurretInCenterToolValue : BOOL
GET
                    bogTurretInCenterToolValue := bogTurretInCenter.Value;

                  
END_GET
END_PROPERTY

PROPERTY bogVehiculeTrainModeToolValue : BOOL
GET
                    bogVehiculeTrainModeToolValue := bogVehiculeTrainMode.Value;

                  
END_GET
END_PROPERTY

PROPERTY bogIncoherenceLateralStopAndKeyToolValue : BOOL
GET
                    bogIncoherenceLateralStopAndKeyToolValue := bogIncoherenceLateralStopAndKey.Value;

                  
END_GET
END_PROPERTY

PROPERTY bogWorkModeToolValue : BOOL
GET
                    bogWorkModeToolValue := bogWorkMode.Value;

                  
END_GET
END_PROPERTY

PROPERTY bogSafetyElectricPumpToolValue : BOOL
GET
                    bogSafetyElectricPumpToolValue := bogSafetyElectricPump.Value;

                  
END_GET
END_PROPERTY

PROPERTY bogDownhill150mmToolValue : BOOL
GET
                    bogDownhill150mmToolValue := bogDownhill150mm.Value;

                  
END_GET
END_PROPERTY

PROPERTY bogTrainModeAllowToolValue : BOOL
GET
                    bogTrainModeAllowToolValue := bogTrainModeAllow.Value;

                  
END_GET
END_PROPERTY

PROPERTY bogBrakeTestServiceToolValue : BOOL
GET
                    bogBrakeTestServiceToolValue := bogBrakeTestService.Value;

                  
END_GET
END_PROPERTY

PROPERTY bogBrakePressureFaultToolValue : BOOL
GET
                    bogBrakePressureFaultToolValue := bogBrakePressureFault.Value;

                  
END_GET
END_PROPERTY

PROPERTY bogActivateMeasuringMastToolValue : BOOL
GET
                    bogActivateMeasuringMastToolValue := bogActivateMeasuringMast.Value;

                  
END_GET
END_PROPERTY

PROPERTY bogAutoMovementDirectionLightToolValue : BOOL
GET
                    bogAutoMovementDirectionLightToolValue := bogAutoMovementDirectionLight.Value;

                  
END_GET
END_PROPERTY

PROPERTY bogBackRailwayAxleLowPositionToolValue : BOOL
GET
                    bogBackRailwayAxleLowPositionToolValue := bogBackRailwayAxleLowPosition.Value;

                  
END_GET
END_PROPERTY

PROPERTY bogFrontRailwayAxleLowPositionToolValue : BOOL
GET
                    bogFrontRailwayAxleLowPositionToolValue := bogFrontRailwayAxleLowPosition.Value;

                  
END_GET
END_PROPERTY

PROPERTY bogBackRailwayAxleServiceBrakeToolValue : BOOL
GET
                    bogBackRailwayAxleServiceBrakeToolValue := bogBackRailwayAxleServiceBrake.Value;

                  
END_GET
END_PROPERTY

PROPERTY bogFrontRailwayAxleServiceBrakeToolValue : BOOL
GET
                    bogFrontRailwayAxleServiceBrakeToolValue := bogFrontRailwayAxleServiceBrake.Value;

                  
END_GET
END_PROPERTY

PROPERTY bogBackRailwayAxleParkBrakeToolValue : BOOL
GET
                    bogBackRailwayAxleParkBrakeToolValue := bogBackRailwayAxleParkBrake.Value;

                  
END_GET
END_PROPERTY

PROPERTY bogFrontRailwayAxleParkBrakeToolValue : BOOL
GET
                    bogFrontRailwayAxleParkBrakeToolValue := bogFrontRailwayAxleParkBrake.Value;

                  
END_GET
END_PROPERTY

PROPERTY bogStatusFrontLeftTrainBrakeTestToolValue : BOOL
GET
                    bogStatusFrontLeftTrainBrakeTestToolValue := bogStatusFrontLeftTrainBrakeTest.Value;

                  
END_GET
END_PROPERTY

PROPERTY bogStatFrontRightTrainBrakeTestToolValue : BOOL
GET
                    bogStatFrontRightTrainBrakeTestToolValue := bogStatFrontRightTrainBrakeTest.Value;

                  
END_GET
END_PROPERTY

PROPERTY bogStatusBackLeftTrainBrakeTestToolValue : BOOL
GET
                    bogStatusBackLeftTrainBrakeTestToolValue := bogStatusBackLeftTrainBrakeTest.Value;

                  
END_GET
END_PROPERTY

PROPERTY bogStatusBackRightTrainBrakeTestToolValue : BOOL
GET
                    bogStatusBackRightTrainBrakeTestToolValue := bogStatusBackRightTrainBrakeTest.Value;

                  
END_GET
END_PROPERTY

PROPERTY bogAlarmAruToolValue : BOOL
GET
                    bogAlarmAruToolValue := bogAlarmAru.Value;

                  
END_GET
END_PROPERTY

PROPERTY bogLitmitSpeedExceededToolValue : BOOL
GET
                    bogLitmitSpeedExceededToolValue := bogLitmitSpeedExceeded.Value;

                  
END_GET
END_PROPERTY

PROPERTY bogShowCameraToolValue : BOOL
GET
                    bogShowCameraToolValue := bogShowCamera.Value;

                  
END_GET
END_PROPERTY

PROPERTY bogFixeAxleFrequencyFaultToolValue : BOOL
GET
                    bogFixeAxleFrequencyFaultToolValue := bogFixeAxleFrequencyFault.Value;

                  
END_GET
END_PROPERTY

PROPERTY bogOscillantAxleFrequencyFaultToolValue : BOOL
GET
                    bogOscillantAxleFrequencyFaultToolValue := bogOscillantAxleFrequencyFault.Value;

                  
END_GET
END_PROPERTY

PROPERTY bogTemperatureTransmAlarmToolValue : BOOL
GET
                    bogTemperatureTransmAlarmToolValue := bogTemperatureTransmAlarm.Value;

                  
END_GET
END_PROPERTY

PROPERTY bogUserCodeOptionToolValue : BOOL
GET
                    bogUserCodeOptionToolValue := bogUserCodeOption.Value;

                  
END_GET
END_PROPERTY

PROPERTY bogRequestForwardTransRailToolValue : BOOL
GET
                    bogRequestForwardTransRailToolValue := bogRequestForwardTransRail.Value;

                  
END_GET
END_PROPERTY

PROPERTY bogRequestBackwardTransRailToolValue : BOOL
GET
                    bogRequestBackwardTransRailToolValue := bogRequestBackwardTransRail.Value;

                  
END_GET
END_PROPERTY

PROPERTY bogEvForwardFaultToolValue : BOOL
GET
                    bogEvForwardFaultToolValue := bogEvForwardFault.Value;

                  
END_GET
END_PROPERTY

PROPERTY bogEvBackwardFaultToolValue : BOOL
GET
                    bogEvBackwardFaultToolValue := bogEvBackwardFault.Value;

                  
END_GET
END_PROPERTY

PROPERTY bogIncoherenceModeTravailToolValue : BOOL
GET
                    bogIncoherenceModeTravailToolValue := bogIncoherenceModeTravail.Value;

                  
END_GET
END_PROPERTY

PROPERTY bogIncoherenceBasketStopAndKeyToolValue : BOOL
GET
                    bogIncoherenceBasketStopAndKeyToolValue := bogIncoherenceBasketStopAndKey.Value;

                  
END_GET
END_PROPERTY

PROPERTY bogCenteredAdvanceJoystickToolValue : BOOL
GET
                    bogCenteredAdvanceJoystickToolValue := bogCenteredAdvanceJoystick.Value;

                  
END_GET
END_PROPERTY

PROPERTY bogKlaxonToolValue : BOOL
GET
                    bogKlaxonToolValue := bogKlaxon.Value;

                  
END_GET
END_PROPERTY

PROPERTY bogGachetteToolValue : BOOL
GET
                    bogGachetteToolValue := bogGachette.Value;

                  
END_GET
END_PROPERTY

PROPERTY bogStopMoteurToolValue : BOOL
GET
                    bogStopMoteurToolValue := bogStopMoteur.Value;

                  
END_GET
END_PROPERTY

PROPERTY bogEStopToolValue : BOOL
GET
                    bogEStopToolValue := bogEStop.Value;

                  
END_GET
END_PROPERTY

PROPERTY bogDeadManToolValue : BOOL
GET
                    bogDeadManToolValue := bogDeadMan.Value;

                  
END_GET
END_PROPERTY

PROPERTY bogSignalDangerModeToolValue : BOOL
GET
                    bogSignalDangerModeToolValue := bogSignalDangerMode.Value;

                  
END_GET
END_PROPERTY

PROPERTY bogLimitSpeedLowSpeedBrakeTestToolValue : BOOL
GET
                    bogLimitSpeedLowSpeedBrakeTestToolValue := bogLimitSpeedLowSpeedBrakeTest.Value;

                  
END_GET
END_PROPERTY

PROPERTY bogSlopeSensorFaultToolValue : BOOL
GET
                    bogSlopeSensorFaultToolValue := bogSlopeSensorFault.Value;

                  
END_GET
END_PROPERTY

PROPERTY bogMastMeasureFaultToolValue : BOOL
GET
                    bogMastMeasureFaultToolValue := bogMastMeasureFault.Value;

                  
END_GET
END_PROPERTY

PROPERTY i16gEncodeurTurretAngleToolValue : INT
GET
                    IF i16gEncodeurTurretAngle.ToolScalingDivisor = 0 OR i16gEncodeurTurretAngle.AppScalingMultiplier = 0 THEN
	_MatchLog^.Error("Get i16gEncodeurTurretAngleToolValue", "Division by Zero!");
	RETURN;
END_IF

i16gEncodeurTurretAngleToolValue := TO_INT(((i16gEncodeurTurretAngle.Value - i16gEncodeurTurretAngle.AppScalingOffset) * i16gEncodeurTurretAngle.AppScalingDivisor / i16gEncodeurTurretAngle.AppScalingMultiplier * i16gEncodeurTurretAngle.ToolScalingMultiplier / i16gEncodeurTurretAngle.ToolScalingDivisor) + i16gEncodeurTurretAngle.ToolScalingOffset);

                  
END_GET
END_PROPERTY

METHOD InitializeCanSignals
                  bogBreak_Parking_On_Off.AppScalingDivisor :=1;
bogBreak_Parking_On_Off.AppScalingMultiplier :=1;
bogBreak_Parking_On_Off.AppScalingOffset :=0;
bogBreak_Parking_On_Off.AppUnit :="";
bogBreak_Parking_On_Off.CanDefault :=0;
bogBreak_Parking_On_Off.CanInit :=0;
bogBreak_Parking_On_Off.CanMax :=1;
bogBreak_Parking_On_Off.CanMin :=0;
bogBreak_Parking_On_Off.CanUnit :="";
bogBreak_Parking_On_Off.Description :="Break Parking Status ";
bogBreak_Parking_On_Off.ErrorReaction := eErrorReaction.ERSIG_DFLT;
bogBreak_Parking_On_Off.ReceiverAdress :=1;
bogBreak_Parking_On_Off.ToolScalingDivisor :=1;
bogBreak_Parking_On_Off.ToolScalingMultiplier :=1;
bogBreak_Parking_On_Off.ToolScalingOffset :=0;
bogBreak_Parking_On_Off.ToolUnit :="";

bogBreak_Faillure_On_Off.AppScalingDivisor :=1;
bogBreak_Faillure_On_Off.AppScalingMultiplier :=1;
bogBreak_Faillure_On_Off.AppScalingOffset :=0;
bogBreak_Faillure_On_Off.AppUnit :="";
bogBreak_Faillure_On_Off.CanDefault :=0;
bogBreak_Faillure_On_Off.CanInit :=0;
bogBreak_Faillure_On_Off.CanMax :=1;
bogBreak_Faillure_On_Off.CanMin :=0;
bogBreak_Faillure_On_Off.CanUnit :="";
bogBreak_Faillure_On_Off.Description :="Break Faillure Status";
bogBreak_Faillure_On_Off.ErrorReaction := eErrorReaction.ERSIG_DFLT;
bogBreak_Faillure_On_Off.ReceiverAdress :=1;
bogBreak_Faillure_On_Off.ToolScalingDivisor :=1;
bogBreak_Faillure_On_Off.ToolScalingMultiplier :=1;
bogBreak_Faillure_On_Off.ToolScalingOffset :=0;
bogBreak_Faillure_On_Off.ToolUnit :="";

bogMovement_Allow_Nacelle.AppScalingDivisor :=1;
bogMovement_Allow_Nacelle.AppScalingMultiplier :=1;
bogMovement_Allow_Nacelle.AppScalingOffset :=0;
bogMovement_Allow_Nacelle.AppUnit :="";
bogMovement_Allow_Nacelle.CanDefault :=0;
bogMovement_Allow_Nacelle.CanInit :=0;
bogMovement_Allow_Nacelle.CanMax :=1;
bogMovement_Allow_Nacelle.CanMin :=0;
bogMovement_Allow_Nacelle.CanUnit :="";
bogMovement_Allow_Nacelle.Description :="Movement Allow Status";
bogMovement_Allow_Nacelle.ErrorReaction := eErrorReaction.ERSIG_DFLT;
bogMovement_Allow_Nacelle.ReceiverAdress :=1;
bogMovement_Allow_Nacelle.ToolScalingDivisor :=1;
bogMovement_Allow_Nacelle.ToolScalingMultiplier :=1;
bogMovement_Allow_Nacelle.ToolScalingOffset :=0;
bogMovement_Allow_Nacelle.ToolUnit :="";

bogTurretSectorInCenter.AppScalingDivisor :=1;
bogTurretSectorInCenter.AppScalingMultiplier :=1;
bogTurretSectorInCenter.AppScalingOffset :=0;
bogTurretSectorInCenter.AppUnit :="";
bogTurretSectorInCenter.CanDefault :=0;
bogTurretSectorInCenter.CanInit :=0;
bogTurretSectorInCenter.CanMax :=1;
bogTurretSectorInCenter.CanMin :=0;
bogTurretSectorInCenter.CanUnit :="";
bogTurretSectorInCenter.Description :="Turret Sector in Center";
bogTurretSectorInCenter.ErrorReaction := eErrorReaction.ERSIG_DFLT;
bogTurretSectorInCenter.ReceiverAdress :=1;
bogTurretSectorInCenter.ToolScalingDivisor :=1;
bogTurretSectorInCenter.ToolScalingMultiplier :=1;
bogTurretSectorInCenter.ToolScalingOffset :=0;
bogTurretSectorInCenter.ToolUnit :="";

bogTurretInCenter.AppScalingDivisor :=1;
bogTurretInCenter.AppScalingMultiplier :=1;
bogTurretInCenter.AppScalingOffset :=0;
bogTurretInCenter.AppUnit :="";
bogTurretInCenter.CanDefault :=0;
bogTurretInCenter.CanInit :=0;
bogTurretInCenter.CanMax :=1;
bogTurretInCenter.CanMin :=0;
bogTurretInCenter.CanUnit :="";
bogTurretInCenter.Description :="Turret in Center";
bogTurretInCenter.ErrorReaction := eErrorReaction.ERSIG_DFLT;
bogTurretInCenter.ReceiverAdress :=1;
bogTurretInCenter.ToolScalingDivisor :=1;
bogTurretInCenter.ToolScalingMultiplier :=1;
bogTurretInCenter.ToolScalingOffset :=0;
bogTurretInCenter.ToolUnit :="";

bogVehiculeTrainMode.AppScalingDivisor :=1;
bogVehiculeTrainMode.AppScalingMultiplier :=1;
bogVehiculeTrainMode.AppScalingOffset :=0;
bogVehiculeTrainMode.AppUnit :="";
bogVehiculeTrainMode.CanDefault :=0;
bogVehiculeTrainMode.CanInit :=0;
bogVehiculeTrainMode.CanMax :=1;
bogVehiculeTrainMode.CanMin :=0;
bogVehiculeTrainMode.CanUnit :="";
bogVehiculeTrainMode.Description :="Vehicule in Train Mode (Speed in MPH)";
bogVehiculeTrainMode.ErrorReaction := eErrorReaction.ERSIG_DFLT;
bogVehiculeTrainMode.ReceiverAdress :=1;
bogVehiculeTrainMode.ToolScalingDivisor :=1;
bogVehiculeTrainMode.ToolScalingMultiplier :=1;
bogVehiculeTrainMode.ToolScalingOffset :=0;
bogVehiculeTrainMode.ToolUnit :="";

bogIncoherenceLateralStopAndKey.AppScalingDivisor :=1;
bogIncoherenceLateralStopAndKey.AppScalingMultiplier :=1;
bogIncoherenceLateralStopAndKey.AppScalingOffset :=0;
bogIncoherenceLateralStopAndKey.AppUnit :="";
bogIncoherenceLateralStopAndKey.CanDefault :=0;
bogIncoherenceLateralStopAndKey.CanInit :=0;
bogIncoherenceLateralStopAndKey.CanMax :=1;
bogIncoherenceLateralStopAndKey.CanMin :=0;
bogIncoherenceLateralStopAndKey.CanUnit :="";
bogIncoherenceLateralStopAndKey.Description :="Incoherence between Lateral Stop and Key selector (A47)";
bogIncoherenceLateralStopAndKey.ErrorReaction := eErrorReaction.ERSIG_DFLT;
bogIncoherenceLateralStopAndKey.ReceiverAdress :=1;
bogIncoherenceLateralStopAndKey.ToolScalingDivisor :=1;
bogIncoherenceLateralStopAndKey.ToolScalingMultiplier :=1;
bogIncoherenceLateralStopAndKey.ToolScalingOffset :=0;
bogIncoherenceLateralStopAndKey.ToolUnit :="";

bogWorkMode.AppScalingDivisor :=1;
bogWorkMode.AppScalingMultiplier :=1;
bogWorkMode.AppScalingOffset :=0;
bogWorkMode.AppUnit :="";
bogWorkMode.CanDefault :=0;
bogWorkMode.CanInit :=0;
bogWorkMode.CanMax :=1;
bogWorkMode.CanMin :=0;
bogWorkMode.CanUnit :="";
bogWorkMode.Description :="0=Work Mode activate 1=Site Acces Mode  (A4)";
bogWorkMode.ErrorReaction := eErrorReaction.ERSIG_DFLT;
bogWorkMode.ReceiverAdress :=1;
bogWorkMode.ToolScalingDivisor :=1;
bogWorkMode.ToolScalingMultiplier :=1;
bogWorkMode.ToolScalingOffset :=0;
bogWorkMode.ToolUnit :="";

bogSafetyElectricPump.AppScalingDivisor :=1;
bogSafetyElectricPump.AppScalingMultiplier :=1;
bogSafetyElectricPump.AppScalingOffset :=0;
bogSafetyElectricPump.AppUnit :="";
bogSafetyElectricPump.CanDefault :=0;
bogSafetyElectricPump.CanInit :=0;
bogSafetyElectricPump.CanMax :=1;
bogSafetyElectricPump.CanMin :=0;
bogSafetyElectricPump.CanUnit :="";
bogSafetyElectricPump.Description :="Safety Electric Pump Activate (A44)";
bogSafetyElectricPump.ErrorReaction := eErrorReaction.ERSIG_DFLT;
bogSafetyElectricPump.ReceiverAdress :=1;
bogSafetyElectricPump.ToolScalingDivisor :=1;
bogSafetyElectricPump.ToolScalingMultiplier :=1;
bogSafetyElectricPump.ToolScalingOffset :=0;
bogSafetyElectricPump.ToolUnit :="";

bogDownhill150mm.AppScalingDivisor :=1;
bogDownhill150mm.AppScalingMultiplier :=1;
bogDownhill150mm.AppScalingOffset :=0;
bogDownhill150mm.AppUnit :="";
bogDownhill150mm.CanDefault :=0;
bogDownhill150mm.CanInit :=0;
bogDownhill150mm.CanMax :=1;
bogDownhill150mm.CanMin :=0;
bogDownhill150mm.CanUnit :="";
bogDownhill150mm.Description :="Downhill between 150mm and 200mm (A13)";
bogDownhill150mm.ErrorReaction := eErrorReaction.ERSIG_DFLT;
bogDownhill150mm.ReceiverAdress :=1;
bogDownhill150mm.ToolScalingDivisor :=1;
bogDownhill150mm.ToolScalingMultiplier :=1;
bogDownhill150mm.ToolScalingOffset :=0;
bogDownhill150mm.ToolUnit :="";

bogTrainModeAllow.AppScalingDivisor :=1;
bogTrainModeAllow.AppScalingMultiplier :=1;
bogTrainModeAllow.AppScalingOffset :=0;
bogTrainModeAllow.AppUnit :="";
bogTrainModeAllow.CanDefault :=0;
bogTrainModeAllow.CanInit :=0;
bogTrainModeAllow.CanMax :=1;
bogTrainModeAllow.CanMin :=0;
bogTrainModeAllow.CanUnit :="";
bogTrainModeAllow.Description :="Train Mode Allow (A10)";
bogTrainModeAllow.ErrorReaction := eErrorReaction.ERSIG_DFLT;
bogTrainModeAllow.ReceiverAdress :=1;
bogTrainModeAllow.ToolScalingDivisor :=1;
bogTrainModeAllow.ToolScalingMultiplier :=1;
bogTrainModeAllow.ToolScalingOffset :=0;
bogTrainModeAllow.ToolUnit :="";

bogBrakeTestService.AppScalingDivisor :=1;
bogBrakeTestService.AppScalingMultiplier :=1;
bogBrakeTestService.AppScalingOffset :=0;
bogBrakeTestService.AppUnit :="";
bogBrakeTestService.CanDefault :=0;
bogBrakeTestService.CanInit :=0;
bogBrakeTestService.CanMax :=1;
bogBrakeTestService.CanMin :=0;
bogBrakeTestService.CanUnit :="";
bogBrakeTestService.Description :="Brake test need to be launch (A22)";
bogBrakeTestService.ErrorReaction := eErrorReaction.ERSIG_DFLT;
bogBrakeTestService.ReceiverAdress :=1;
bogBrakeTestService.ToolScalingDivisor :=1;
bogBrakeTestService.ToolScalingMultiplier :=1;
bogBrakeTestService.ToolScalingOffset :=0;
bogBrakeTestService.ToolUnit :="";

bogBrakePressureFault.AppScalingDivisor :=1;
bogBrakePressureFault.AppScalingMultiplier :=1;
bogBrakePressureFault.AppScalingOffset :=0;
bogBrakePressureFault.AppUnit :="";
bogBrakePressureFault.CanDefault :=0;
bogBrakePressureFault.CanInit :=0;
bogBrakePressureFault.CanMax :=1;
bogBrakePressureFault.CanMin :=0;
bogBrakePressureFault.CanUnit :="";
bogBrakePressureFault.Description :="Brake Pressure Fault (A14)";
bogBrakePressureFault.ErrorReaction := eErrorReaction.ERSIG_DFLT;
bogBrakePressureFault.ReceiverAdress :=1;
bogBrakePressureFault.ToolScalingDivisor :=1;
bogBrakePressureFault.ToolScalingMultiplier :=1;
bogBrakePressureFault.ToolScalingOffset :=0;
bogBrakePressureFault.ToolUnit :="";

bogActivateMeasuringMast.AppScalingDivisor :=1;
bogActivateMeasuringMast.AppScalingMultiplier :=1;
bogActivateMeasuringMast.AppScalingOffset :=0;
bogActivateMeasuringMast.AppUnit :="";
bogActivateMeasuringMast.CanDefault :=0;
bogActivateMeasuringMast.CanInit :=0;
bogActivateMeasuringMast.CanMax :=1;
bogActivateMeasuringMast.CanMin :=0;
bogActivateMeasuringMast.CanUnit :="";
bogActivateMeasuringMast.Description :="Activate Measuring Mast (A21)";
bogActivateMeasuringMast.ErrorReaction := eErrorReaction.ERSIG_DFLT;
bogActivateMeasuringMast.ReceiverAdress :=1;
bogActivateMeasuringMast.ToolScalingDivisor :=1;
bogActivateMeasuringMast.ToolScalingMultiplier :=1;
bogActivateMeasuringMast.ToolScalingOffset :=0;
bogActivateMeasuringMast.ToolUnit :="";

bogAutoMovementDirectionLight.AppScalingDivisor :=1;
bogAutoMovementDirectionLight.AppScalingMultiplier :=1;
bogAutoMovementDirectionLight.AppScalingOffset :=0;
bogAutoMovementDirectionLight.AppUnit :="";
bogAutoMovementDirectionLight.CanDefault :=0;
bogAutoMovementDirectionLight.CanInit :=0;
bogAutoMovementDirectionLight.CanMax :=1;
bogAutoMovementDirectionLight.CanMin :=0;
bogAutoMovementDirectionLight.CanUnit :="";
bogAutoMovementDirectionLight.Description :="Auto Movement Direction Light (A23)";
bogAutoMovementDirectionLight.ErrorReaction := eErrorReaction.ERSIG_DFLT;
bogAutoMovementDirectionLight.ReceiverAdress :=1;
bogAutoMovementDirectionLight.ToolScalingDivisor :=1;
bogAutoMovementDirectionLight.ToolScalingMultiplier :=1;
bogAutoMovementDirectionLight.ToolScalingOffset :=0;
bogAutoMovementDirectionLight.ToolUnit :="";

bogBackRailwayAxleLowPosition.AppScalingDivisor :=1;
bogBackRailwayAxleLowPosition.AppScalingMultiplier :=1;
bogBackRailwayAxleLowPosition.AppScalingOffset :=0;
bogBackRailwayAxleLowPosition.AppUnit :="";
bogBackRailwayAxleLowPosition.CanDefault :=0;
bogBackRailwayAxleLowPosition.CanInit :=0;
bogBackRailwayAxleLowPosition.CanMax :=1;
bogBackRailwayAxleLowPosition.CanMin :=0;
bogBackRailwayAxleLowPosition.CanUnit :="";
bogBackRailwayAxleLowPosition.Description :="Back Railway Axle in Low Position (A7)";
bogBackRailwayAxleLowPosition.ErrorReaction := eErrorReaction.ERSIG_DFLT;
bogBackRailwayAxleLowPosition.ReceiverAdress :=1;
bogBackRailwayAxleLowPosition.ToolScalingDivisor :=1;
bogBackRailwayAxleLowPosition.ToolScalingMultiplier :=1;
bogBackRailwayAxleLowPosition.ToolScalingOffset :=0;
bogBackRailwayAxleLowPosition.ToolUnit :="";

bogFrontRailwayAxleLowPosition.AppScalingDivisor :=1;
bogFrontRailwayAxleLowPosition.AppScalingMultiplier :=1;
bogFrontRailwayAxleLowPosition.AppScalingOffset :=0;
bogFrontRailwayAxleLowPosition.AppUnit :="";
bogFrontRailwayAxleLowPosition.CanDefault :=0;
bogFrontRailwayAxleLowPosition.CanInit :=0;
bogFrontRailwayAxleLowPosition.CanMax :=1;
bogFrontRailwayAxleLowPosition.CanMin :=0;
bogFrontRailwayAxleLowPosition.CanUnit :="";
bogFrontRailwayAxleLowPosition.Description :="Front Railway Axle in Low Position (A7)";
bogFrontRailwayAxleLowPosition.ErrorReaction := eErrorReaction.ERSIG_DFLT;
bogFrontRailwayAxleLowPosition.ReceiverAdress :=1;
bogFrontRailwayAxleLowPosition.ToolScalingDivisor :=1;
bogFrontRailwayAxleLowPosition.ToolScalingMultiplier :=1;
bogFrontRailwayAxleLowPosition.ToolScalingOffset :=0;
bogFrontRailwayAxleLowPosition.ToolUnit :="";

bogBackRailwayAxleServiceBrake.AppScalingDivisor :=1;
bogBackRailwayAxleServiceBrake.AppScalingMultiplier :=1;
bogBackRailwayAxleServiceBrake.AppScalingOffset :=0;
bogBackRailwayAxleServiceBrake.AppUnit :="";
bogBackRailwayAxleServiceBrake.CanDefault :=0;
bogBackRailwayAxleServiceBrake.CanInit :=0;
bogBackRailwayAxleServiceBrake.CanMax :=1;
bogBackRailwayAxleServiceBrake.CanMin :=0;
bogBackRailwayAxleServiceBrake.CanUnit :="";
bogBackRailwayAxleServiceBrake.Description :="Back Railway Axle Service Brake (A25)";
bogBackRailwayAxleServiceBrake.ErrorReaction := eErrorReaction.ERSIG_DFLT;
bogBackRailwayAxleServiceBrake.ReceiverAdress :=1;
bogBackRailwayAxleServiceBrake.ToolScalingDivisor :=1;
bogBackRailwayAxleServiceBrake.ToolScalingMultiplier :=1;
bogBackRailwayAxleServiceBrake.ToolScalingOffset :=0;
bogBackRailwayAxleServiceBrake.ToolUnit :="";

bogFrontRailwayAxleServiceBrake.AppScalingDivisor :=1;
bogFrontRailwayAxleServiceBrake.AppScalingMultiplier :=1;
bogFrontRailwayAxleServiceBrake.AppScalingOffset :=0;
bogFrontRailwayAxleServiceBrake.AppUnit :="";
bogFrontRailwayAxleServiceBrake.CanDefault :=0;
bogFrontRailwayAxleServiceBrake.CanInit :=0;
bogFrontRailwayAxleServiceBrake.CanMax :=1;
bogFrontRailwayAxleServiceBrake.CanMin :=0;
bogFrontRailwayAxleServiceBrake.CanUnit :="";
bogFrontRailwayAxleServiceBrake.Description :="Front Railway Axle Service Brake (A25)";
bogFrontRailwayAxleServiceBrake.ErrorReaction := eErrorReaction.ERSIG_DFLT;
bogFrontRailwayAxleServiceBrake.ReceiverAdress :=1;
bogFrontRailwayAxleServiceBrake.ToolScalingDivisor :=1;
bogFrontRailwayAxleServiceBrake.ToolScalingMultiplier :=1;
bogFrontRailwayAxleServiceBrake.ToolScalingOffset :=0;
bogFrontRailwayAxleServiceBrake.ToolUnit :="";

bogBackRailwayAxleParkBrake.AppScalingDivisor :=1;
bogBackRailwayAxleParkBrake.AppScalingMultiplier :=1;
bogBackRailwayAxleParkBrake.AppScalingOffset :=0;
bogBackRailwayAxleParkBrake.AppUnit :="";
bogBackRailwayAxleParkBrake.CanDefault :=0;
bogBackRailwayAxleParkBrake.CanInit :=0;
bogBackRailwayAxleParkBrake.CanMax :=1;
bogBackRailwayAxleParkBrake.CanMin :=0;
bogBackRailwayAxleParkBrake.CanUnit :="";
bogBackRailwayAxleParkBrake.Description :="Back Railway Axle Park Brake (A26)";
bogBackRailwayAxleParkBrake.ErrorReaction := eErrorReaction.ERSIG_DFLT;
bogBackRailwayAxleParkBrake.ReceiverAdress :=1;
bogBackRailwayAxleParkBrake.ToolScalingDivisor :=1;
bogBackRailwayAxleParkBrake.ToolScalingMultiplier :=1;
bogBackRailwayAxleParkBrake.ToolScalingOffset :=0;
bogBackRailwayAxleParkBrake.ToolUnit :="";

bogFrontRailwayAxleParkBrake.AppScalingDivisor :=1;
bogFrontRailwayAxleParkBrake.AppScalingMultiplier :=1;
bogFrontRailwayAxleParkBrake.AppScalingOffset :=0;
bogFrontRailwayAxleParkBrake.AppUnit :="";
bogFrontRailwayAxleParkBrake.CanDefault :=0;
bogFrontRailwayAxleParkBrake.CanInit :=0;
bogFrontRailwayAxleParkBrake.CanMax :=1;
bogFrontRailwayAxleParkBrake.CanMin :=0;
bogFrontRailwayAxleParkBrake.CanUnit :="";
bogFrontRailwayAxleParkBrake.Description :="Front Railway Axle Park Brake (A26) ";
bogFrontRailwayAxleParkBrake.ErrorReaction := eErrorReaction.ERSIG_DFLT;
bogFrontRailwayAxleParkBrake.ReceiverAdress :=1;
bogFrontRailwayAxleParkBrake.ToolScalingDivisor :=1;
bogFrontRailwayAxleParkBrake.ToolScalingMultiplier :=1;
bogFrontRailwayAxleParkBrake.ToolScalingOffset :=0;
bogFrontRailwayAxleParkBrake.ToolUnit :="";

bogStatusFrontLeftTrainBrakeTest.AppScalingDivisor :=1;
bogStatusFrontLeftTrainBrakeTest.AppScalingMultiplier :=1;
bogStatusFrontLeftTrainBrakeTest.AppScalingOffset :=0;
bogStatusFrontLeftTrainBrakeTest.AppUnit :="";
bogStatusFrontLeftTrainBrakeTest.CanDefault :=0;
bogStatusFrontLeftTrainBrakeTest.CanInit :=0;
bogStatusFrontLeftTrainBrakeTest.CanMax :=1;
bogStatusFrontLeftTrainBrakeTest.CanMin :=0;
bogStatusFrontLeftTrainBrakeTest.CanUnit :="";
bogStatusFrontLeftTrainBrakeTest.Description :="Status of Front Left Train Brake Test (A27)";
bogStatusFrontLeftTrainBrakeTest.ErrorReaction := eErrorReaction.ERSIG_DFLT;
bogStatusFrontLeftTrainBrakeTest.ReceiverAdress :=1;
bogStatusFrontLeftTrainBrakeTest.ToolScalingDivisor :=1;
bogStatusFrontLeftTrainBrakeTest.ToolScalingMultiplier :=1;
bogStatusFrontLeftTrainBrakeTest.ToolScalingOffset :=0;
bogStatusFrontLeftTrainBrakeTest.ToolUnit :="";

bogStatFrontRightTrainBrakeTest.AppScalingDivisor :=1;
bogStatFrontRightTrainBrakeTest.AppScalingMultiplier :=1;
bogStatFrontRightTrainBrakeTest.AppScalingOffset :=0;
bogStatFrontRightTrainBrakeTest.AppUnit :="";
bogStatFrontRightTrainBrakeTest.CanDefault :=0;
bogStatFrontRightTrainBrakeTest.CanInit :=0;
bogStatFrontRightTrainBrakeTest.CanMax :=1;
bogStatFrontRightTrainBrakeTest.CanMin :=0;
bogStatFrontRightTrainBrakeTest.CanUnit :="";
bogStatFrontRightTrainBrakeTest.Description :="Status of Front Right Train Brake Test (A27)";
bogStatFrontRightTrainBrakeTest.ErrorReaction := eErrorReaction.ERSIG_DFLT;
bogStatFrontRightTrainBrakeTest.ReceiverAdress :=1;
bogStatFrontRightTrainBrakeTest.ToolScalingDivisor :=1;
bogStatFrontRightTrainBrakeTest.ToolScalingMultiplier :=1;
bogStatFrontRightTrainBrakeTest.ToolScalingOffset :=0;
bogStatFrontRightTrainBrakeTest.ToolUnit :="";

bogStatusBackLeftTrainBrakeTest.AppScalingDivisor :=1;
bogStatusBackLeftTrainBrakeTest.AppScalingMultiplier :=1;
bogStatusBackLeftTrainBrakeTest.AppScalingOffset :=0;
bogStatusBackLeftTrainBrakeTest.AppUnit :="";
bogStatusBackLeftTrainBrakeTest.CanDefault :=0;
bogStatusBackLeftTrainBrakeTest.CanInit :=0;
bogStatusBackLeftTrainBrakeTest.CanMax :=1;
bogStatusBackLeftTrainBrakeTest.CanMin :=0;
bogStatusBackLeftTrainBrakeTest.CanUnit :="";
bogStatusBackLeftTrainBrakeTest.Description :="Status of Back Left Train Brake Test (A27)";
bogStatusBackLeftTrainBrakeTest.ErrorReaction := eErrorReaction.ERSIG_DFLT;
bogStatusBackLeftTrainBrakeTest.ReceiverAdress :=1;
bogStatusBackLeftTrainBrakeTest.ToolScalingDivisor :=1;
bogStatusBackLeftTrainBrakeTest.ToolScalingMultiplier :=1;
bogStatusBackLeftTrainBrakeTest.ToolScalingOffset :=0;
bogStatusBackLeftTrainBrakeTest.ToolUnit :="";

bogStatusBackRightTrainBrakeTest.AppScalingDivisor :=1;
bogStatusBackRightTrainBrakeTest.AppScalingMultiplier :=1;
bogStatusBackRightTrainBrakeTest.AppScalingOffset :=0;
bogStatusBackRightTrainBrakeTest.AppUnit :="";
bogStatusBackRightTrainBrakeTest.CanDefault :=0;
bogStatusBackRightTrainBrakeTest.CanInit :=0;
bogStatusBackRightTrainBrakeTest.CanMax :=1;
bogStatusBackRightTrainBrakeTest.CanMin :=0;
bogStatusBackRightTrainBrakeTest.CanUnit :="";
bogStatusBackRightTrainBrakeTest.Description :="Status of Back Left Train Brake Test (A27)";
bogStatusBackRightTrainBrakeTest.ErrorReaction := eErrorReaction.ERSIG_DFLT;
bogStatusBackRightTrainBrakeTest.ReceiverAdress :=1;
bogStatusBackRightTrainBrakeTest.ToolScalingDivisor :=1;
bogStatusBackRightTrainBrakeTest.ToolScalingMultiplier :=1;
bogStatusBackRightTrainBrakeTest.ToolScalingOffset :=0;
bogStatusBackRightTrainBrakeTest.ToolUnit :="";

bogAlarmAru.AppScalingDivisor :=1;
bogAlarmAru.AppScalingMultiplier :=1;
bogAlarmAru.AppScalingOffset :=0;
bogAlarmAru.AppUnit :="";
bogAlarmAru.CanDefault :=0;
bogAlarmAru.CanInit :=0;
bogAlarmAru.CanMax :=1;
bogAlarmAru.CanMin :=0;
bogAlarmAru.CanUnit :="";
bogAlarmAru.Description :="Status of the ARU alarm";
bogAlarmAru.ErrorReaction := eErrorReaction.ERSIG_DFLT;
bogAlarmAru.ReceiverAdress :=1;
bogAlarmAru.ToolScalingDivisor :=1;
bogAlarmAru.ToolScalingMultiplier :=1;
bogAlarmAru.ToolScalingOffset :=0;
bogAlarmAru.ToolUnit :="";

bogLitmitSpeedExceeded.AppScalingDivisor :=1;
bogLitmitSpeedExceeded.AppScalingMultiplier :=1;
bogLitmitSpeedExceeded.AppScalingOffset :=0;
bogLitmitSpeedExceeded.AppUnit :="";
bogLitmitSpeedExceeded.CanDefault :=0;
bogLitmitSpeedExceeded.CanInit :=0;
bogLitmitSpeedExceeded.CanMax :=1;
bogLitmitSpeedExceeded.CanMin :=0;
bogLitmitSpeedExceeded.CanUnit :="";
bogLitmitSpeedExceeded.Description :="Flag when limit speed is exceeded";
bogLitmitSpeedExceeded.ErrorReaction := eErrorReaction.ERSIG_DFLT;
bogLitmitSpeedExceeded.ReceiverAdress :=1;
bogLitmitSpeedExceeded.ToolScalingDivisor :=1;
bogLitmitSpeedExceeded.ToolScalingMultiplier :=1;
bogLitmitSpeedExceeded.ToolScalingOffset :=0;
bogLitmitSpeedExceeded.ToolUnit :="";

bogShowCamera.AppScalingDivisor :=1;
bogShowCamera.AppScalingMultiplier :=1;
bogShowCamera.AppScalingOffset :=0;
bogShowCamera.AppUnit :="";
bogShowCamera.CanDefault :=0;
bogShowCamera.CanInit :=0;
bogShowCamera.CanMax :=1;
bogShowCamera.CanMin :=0;
bogShowCamera.CanUnit :="";
bogShowCamera.Description :="Display camera on screen when translation is solicited";
bogShowCamera.ErrorReaction := eErrorReaction.ERSIG_DFLT;
bogShowCamera.ReceiverAdress :=1;
bogShowCamera.ToolScalingDivisor :=1;
bogShowCamera.ToolScalingMultiplier :=1;
bogShowCamera.ToolScalingOffset :=0;
bogShowCamera.ToolUnit :="";

bogFixeAxleFrequencyFault.AppScalingDivisor :=1;
bogFixeAxleFrequencyFault.AppScalingMultiplier :=1;
bogFixeAxleFrequencyFault.AppScalingOffset :=0;
bogFixeAxleFrequencyFault.AppUnit :="";
bogFixeAxleFrequencyFault.CanDefault :=0;
bogFixeAxleFrequencyFault.CanInit :=0;
bogFixeAxleFrequencyFault.CanMax :=1;
bogFixeAxleFrequencyFault.CanMin :=0;
bogFixeAxleFrequencyFault.CanUnit :="";
bogFixeAxleFrequencyFault.Description :="Fixed axle Speed sensor 2 fault";
bogFixeAxleFrequencyFault.ErrorReaction := eErrorReaction.ERSIG_DFLT;
bogFixeAxleFrequencyFault.ReceiverAdress :=1;
bogFixeAxleFrequencyFault.ToolScalingDivisor :=1;
bogFixeAxleFrequencyFault.ToolScalingMultiplier :=1;
bogFixeAxleFrequencyFault.ToolScalingOffset :=0;
bogFixeAxleFrequencyFault.ToolUnit :="";

bogOscillantAxleFrequencyFault.AppScalingDivisor :=1;
bogOscillantAxleFrequencyFault.AppScalingMultiplier :=1;
bogOscillantAxleFrequencyFault.AppScalingOffset :=0;
bogOscillantAxleFrequencyFault.AppUnit :="";
bogOscillantAxleFrequencyFault.CanDefault :=0;
bogOscillantAxleFrequencyFault.CanInit :=0;
bogOscillantAxleFrequencyFault.CanMax :=1;
bogOscillantAxleFrequencyFault.CanMin :=0;
bogOscillantAxleFrequencyFault.CanUnit :="";
bogOscillantAxleFrequencyFault.Description :="Fixed axle Speed sensor 1 fault";
bogOscillantAxleFrequencyFault.ErrorReaction := eErrorReaction.ERSIG_DFLT;
bogOscillantAxleFrequencyFault.ReceiverAdress :=1;
bogOscillantAxleFrequencyFault.ToolScalingDivisor :=1;
bogOscillantAxleFrequencyFault.ToolScalingMultiplier :=1;
bogOscillantAxleFrequencyFault.ToolScalingOffset :=0;
bogOscillantAxleFrequencyFault.ToolUnit :="";

bogTemperatureTransmAlarm.AppScalingDivisor :=1;
bogTemperatureTransmAlarm.AppScalingMultiplier :=1;
bogTemperatureTransmAlarm.AppScalingOffset :=0;
bogTemperatureTransmAlarm.AppUnit :="";
bogTemperatureTransmAlarm.CanDefault :=0;
bogTemperatureTransmAlarm.CanInit :=0;
bogTemperatureTransmAlarm.CanMax :=1;
bogTemperatureTransmAlarm.CanMin :=0;
bogTemperatureTransmAlarm.CanUnit :="";
bogTemperatureTransmAlarm.Description :="Oil temperature alarm";
bogTemperatureTransmAlarm.ErrorReaction := eErrorReaction.ERSIG_DFLT;
bogTemperatureTransmAlarm.ReceiverAdress :=1;
bogTemperatureTransmAlarm.ToolScalingDivisor :=1;
bogTemperatureTransmAlarm.ToolScalingMultiplier :=1;
bogTemperatureTransmAlarm.ToolScalingOffset :=0;
bogTemperatureTransmAlarm.ToolUnit :="";

bogUserCodeOption.AppScalingDivisor :=1;
bogUserCodeOption.AppScalingMultiplier :=1;
bogUserCodeOption.AppScalingOffset :=0;
bogUserCodeOption.AppUnit :="";
bogUserCodeOption.CanDefault :=0;
bogUserCodeOption.CanInit :=0;
bogUserCodeOption.CanMax :=1;
bogUserCodeOption.CanMin :=0;
bogUserCodeOption.CanUnit :="";
bogUserCodeOption.Description :="Option user code active";
bogUserCodeOption.ErrorReaction := eErrorReaction.ERSIG_DFLT;
bogUserCodeOption.ReceiverAdress :=1;
bogUserCodeOption.ToolScalingDivisor :=1;
bogUserCodeOption.ToolScalingMultiplier :=1;
bogUserCodeOption.ToolScalingOffset :=0;
bogUserCodeOption.ToolUnit :="";

bogRequestForwardTransRail.AppScalingDivisor :=1;
bogRequestForwardTransRail.AppScalingMultiplier :=1;
bogRequestForwardTransRail.AppScalingOffset :=0;
bogRequestForwardTransRail.AppUnit :="";
bogRequestForwardTransRail.CanDefault :=0;
bogRequestForwardTransRail.CanInit :=0;
bogRequestForwardTransRail.CanMax :=1;
bogRequestForwardTransRail.CanMin :=0;
bogRequestForwardTransRail.CanUnit :="";
bogRequestForwardTransRail.Description :="Request joystick forward trans rail";
bogRequestForwardTransRail.ErrorReaction := eErrorReaction.ERSIG_DFLT;
bogRequestForwardTransRail.ReceiverAdress :=1;
bogRequestForwardTransRail.ToolScalingDivisor :=1;
bogRequestForwardTransRail.ToolScalingMultiplier :=1;
bogRequestForwardTransRail.ToolScalingOffset :=0;
bogRequestForwardTransRail.ToolUnit :="";

bogRequestBackwardTransRail.AppScalingDivisor :=1;
bogRequestBackwardTransRail.AppScalingMultiplier :=1;
bogRequestBackwardTransRail.AppScalingOffset :=0;
bogRequestBackwardTransRail.AppUnit :="";
bogRequestBackwardTransRail.CanDefault :=0;
bogRequestBackwardTransRail.CanInit :=0;
bogRequestBackwardTransRail.CanMax :=1;
bogRequestBackwardTransRail.CanMin :=0;
bogRequestBackwardTransRail.CanUnit :="";
bogRequestBackwardTransRail.Description :="Request joystick forward trans rail";
bogRequestBackwardTransRail.ErrorReaction := eErrorReaction.ERSIG_DFLT;
bogRequestBackwardTransRail.ReceiverAdress :=1;
bogRequestBackwardTransRail.ToolScalingDivisor :=1;
bogRequestBackwardTransRail.ToolScalingMultiplier :=1;
bogRequestBackwardTransRail.ToolScalingOffset :=0;
bogRequestBackwardTransRail.ToolUnit :="";

bogEvForwardFault.AppScalingDivisor :=1;
bogEvForwardFault.AppScalingMultiplier :=1;
bogEvForwardFault.AppScalingOffset :=0;
bogEvForwardFault.AppUnit :="";
bogEvForwardFault.CanDefault :=0;
bogEvForwardFault.CanInit :=0;
bogEvForwardFault.CanMax :=1;
bogEvForwardFault.CanMin :=0;
bogEvForwardFault.CanUnit :="";
bogEvForwardFault.Description :="Ev Forward Fault CC CO";
bogEvForwardFault.ErrorReaction := eErrorReaction.ERSIG_DFLT;
bogEvForwardFault.ReceiverAdress :=1;
bogEvForwardFault.ToolScalingDivisor :=1;
bogEvForwardFault.ToolScalingMultiplier :=1;
bogEvForwardFault.ToolScalingOffset :=0;
bogEvForwardFault.ToolUnit :="";

bogEvBackwardFault.AppScalingDivisor :=1;
bogEvBackwardFault.AppScalingMultiplier :=1;
bogEvBackwardFault.AppScalingOffset :=0;
bogEvBackwardFault.AppUnit :="";
bogEvBackwardFault.CanDefault :=0;
bogEvBackwardFault.CanInit :=0;
bogEvBackwardFault.CanMax :=1;
bogEvBackwardFault.CanMin :=0;
bogEvBackwardFault.CanUnit :="";
bogEvBackwardFault.Description :="Ev Backward Fault CC CO";
bogEvBackwardFault.ErrorReaction := eErrorReaction.ERSIG_DFLT;
bogEvBackwardFault.ReceiverAdress :=1;
bogEvBackwardFault.ToolScalingDivisor :=1;
bogEvBackwardFault.ToolScalingMultiplier :=1;
bogEvBackwardFault.ToolScalingOffset :=0;
bogEvBackwardFault.ToolUnit :="";

bogIncoherenceModeTravail.AppScalingDivisor :=1;
bogIncoherenceModeTravail.AppScalingMultiplier :=1;
bogIncoherenceModeTravail.AppScalingOffset :=0;
bogIncoherenceModeTravail.AppUnit :="";
bogIncoherenceModeTravail.CanDefault :=0;
bogIncoherenceModeTravail.CanInit :=0;
bogIncoherenceModeTravail.CanMax :=1;
bogIncoherenceModeTravail.CanMin :=0;
bogIncoherenceModeTravail.CanUnit :="";
bogIncoherenceModeTravail.Description :="Incoherence between Lateral/Basket Stop and Key selector ";
bogIncoherenceModeTravail.ErrorReaction := eErrorReaction.ERSIG_DFLT;
bogIncoherenceModeTravail.ReceiverAdress :=1;
bogIncoherenceModeTravail.ToolScalingDivisor :=1;
bogIncoherenceModeTravail.ToolScalingMultiplier :=1;
bogIncoherenceModeTravail.ToolScalingOffset :=0;
bogIncoherenceModeTravail.ToolUnit :="";

bogIncoherenceBasketStopAndKey.AppScalingDivisor :=1;
bogIncoherenceBasketStopAndKey.AppScalingMultiplier :=1;
bogIncoherenceBasketStopAndKey.AppScalingOffset :=0;
bogIncoherenceBasketStopAndKey.AppUnit :="";
bogIncoherenceBasketStopAndKey.CanDefault :=0;
bogIncoherenceBasketStopAndKey.CanInit :=0;
bogIncoherenceBasketStopAndKey.CanMax :=1;
bogIncoherenceBasketStopAndKey.CanMin :=0;
bogIncoherenceBasketStopAndKey.CanUnit :="";
bogIncoherenceBasketStopAndKey.Description :="Incoherence between Basket Stop and Key selector";
bogIncoherenceBasketStopAndKey.ErrorReaction := eErrorReaction.ERSIG_DFLT;
bogIncoherenceBasketStopAndKey.ReceiverAdress :=1;
bogIncoherenceBasketStopAndKey.ToolScalingDivisor :=1;
bogIncoherenceBasketStopAndKey.ToolScalingMultiplier :=1;
bogIncoherenceBasketStopAndKey.ToolScalingOffset :=0;
bogIncoherenceBasketStopAndKey.ToolUnit :="";

bogCenteredAdvanceJoystick.AppScalingDivisor :=1;
bogCenteredAdvanceJoystick.AppScalingMultiplier :=1;
bogCenteredAdvanceJoystick.AppScalingOffset :=0;
bogCenteredAdvanceJoystick.AppUnit :="";
bogCenteredAdvanceJoystick.CanDefault :=0;
bogCenteredAdvanceJoystick.CanInit :=0;
bogCenteredAdvanceJoystick.CanMax :=1;
bogCenteredAdvanceJoystick.CanMin :=0;
bogCenteredAdvanceJoystick.CanUnit :="";
bogCenteredAdvanceJoystick.Description :="Advance joystick centered";
bogCenteredAdvanceJoystick.ErrorReaction := eErrorReaction.ERSIG_DFLT;
bogCenteredAdvanceJoystick.ReceiverAdress :=1;
bogCenteredAdvanceJoystick.ToolScalingDivisor :=1;
bogCenteredAdvanceJoystick.ToolScalingMultiplier :=1;
bogCenteredAdvanceJoystick.ToolScalingOffset :=0;
bogCenteredAdvanceJoystick.ToolUnit :="";

bogKlaxon.AppScalingDivisor :=1;
bogKlaxon.AppScalingMultiplier :=1;
bogKlaxon.AppScalingOffset :=0;
bogKlaxon.AppUnit :="";
bogKlaxon.CanDefault :=0;
bogKlaxon.CanInit :=0;
bogKlaxon.CanMax :=1;
bogKlaxon.CanMin :=0;
bogKlaxon.CanUnit :="";
bogKlaxon.Description :="Klaxon";
bogKlaxon.ErrorReaction := eErrorReaction.ERSIG_DFLT;
bogKlaxon.ReceiverAdress :=1;
bogKlaxon.ToolScalingDivisor :=1;
bogKlaxon.ToolScalingMultiplier :=1;
bogKlaxon.ToolScalingOffset :=0;
bogKlaxon.ToolUnit :="";

bogGachette.AppScalingDivisor :=1;
bogGachette.AppScalingMultiplier :=1;
bogGachette.AppScalingOffset :=0;
bogGachette.AppUnit :="";
bogGachette.CanDefault :=0;
bogGachette.CanInit :=0;
bogGachette.CanMax :=1;
bogGachette.CanMin :=0;
bogGachette.CanUnit :="";
bogGachette.Description :="Gachette";
bogGachette.ErrorReaction := eErrorReaction.ERSIG_DFLT;
bogGachette.ReceiverAdress :=1;
bogGachette.ToolScalingDivisor :=1;
bogGachette.ToolScalingMultiplier :=1;
bogGachette.ToolScalingOffset :=0;
bogGachette.ToolUnit :="";

bogStopMoteur.AppScalingDivisor :=1;
bogStopMoteur.AppScalingMultiplier :=1;
bogStopMoteur.AppScalingOffset :=0;
bogStopMoteur.AppUnit :="";
bogStopMoteur.CanDefault :=0;
bogStopMoteur.CanInit :=0;
bogStopMoteur.CanMax :=1;
bogStopMoteur.CanMin :=0;
bogStopMoteur.CanUnit :="";
bogStopMoteur.Description :="BP STOP";
bogStopMoteur.ErrorReaction := eErrorReaction.ERSIG_DFLT;
bogStopMoteur.ReceiverAdress :=1;
bogStopMoteur.ToolScalingDivisor :=1;
bogStopMoteur.ToolScalingMultiplier :=1;
bogStopMoteur.ToolScalingOffset :=0;
bogStopMoteur.ToolUnit :="";

bogEStop.AppScalingDivisor :=1;
bogEStop.AppScalingMultiplier :=1;
bogEStop.AppScalingOffset :=0;
bogEStop.AppUnit :="";
bogEStop.CanDefault :=0;
bogEStop.CanInit :=0;
bogEStop.CanMax :=1;
bogEStop.CanMin :=0;
bogEStop.CanUnit :="";
bogEStop.Description :="Emergency stop";
bogEStop.ErrorReaction := eErrorReaction.ERSIG_DFLT;
bogEStop.ReceiverAdress :=1;
bogEStop.ToolScalingDivisor :=1;
bogEStop.ToolScalingMultiplier :=1;
bogEStop.ToolScalingOffset :=0;
bogEStop.ToolUnit :="";

bogDeadMan.AppScalingDivisor :=1;
bogDeadMan.AppScalingMultiplier :=1;
bogDeadMan.AppScalingOffset :=0;
bogDeadMan.AppUnit :="";
bogDeadMan.CanDefault :=0;
bogDeadMan.CanInit :=0;
bogDeadMan.CanMax :=1;
bogDeadMan.CanMin :=0;
bogDeadMan.CanUnit :="";
bogDeadMan.Description :="Dead man pedal";
bogDeadMan.ErrorReaction := eErrorReaction.ERSIG_DFLT;
bogDeadMan.ReceiverAdress :=1;
bogDeadMan.ToolScalingDivisor :=1;
bogDeadMan.ToolScalingMultiplier :=1;
bogDeadMan.ToolScalingOffset :=0;
bogDeadMan.ToolUnit :="";

bogSignalDangerMode.AppScalingDivisor :=1;
bogSignalDangerMode.AppScalingMultiplier :=1;
bogSignalDangerMode.AppScalingOffset :=0;
bogSignalDangerMode.AppUnit :="";
bogSignalDangerMode.CanDefault :=0;
bogSignalDangerMode.CanInit :=0;
bogSignalDangerMode.CanMax :=1;
bogSignalDangerMode.CanMin :=0;
bogSignalDangerMode.CanUnit :="";
bogSignalDangerMode.Description :="Signal Danger Lights mode";
bogSignalDangerMode.ErrorReaction := eErrorReaction.ERSIG_DFLT;
bogSignalDangerMode.ReceiverAdress :=1;
bogSignalDangerMode.ToolScalingDivisor :=1;
bogSignalDangerMode.ToolScalingMultiplier :=1;
bogSignalDangerMode.ToolScalingOffset :=0;
bogSignalDangerMode.ToolUnit :="";

bogLimitSpeedLowSpeedBrakeTest.AppScalingDivisor :=1;
bogLimitSpeedLowSpeedBrakeTest.AppScalingMultiplier :=1;
bogLimitSpeedLowSpeedBrakeTest.AppScalingOffset :=0;
bogLimitSpeedLowSpeedBrakeTest.AppUnit :="";
bogLimitSpeedLowSpeedBrakeTest.CanDefault :=0;
bogLimitSpeedLowSpeedBrakeTest.CanInit :=0;
bogLimitSpeedLowSpeedBrakeTest.CanMax :=1;
bogLimitSpeedLowSpeedBrakeTest.CanMin :=0;
bogLimitSpeedLowSpeedBrakeTest.CanUnit :="";
bogLimitSpeedLowSpeedBrakeTest.Description :="Limit/low Speed because of none Brake test";
bogLimitSpeedLowSpeedBrakeTest.ErrorReaction := eErrorReaction.ERSIG_DFLT;
bogLimitSpeedLowSpeedBrakeTest.ReceiverAdress :=1;
bogLimitSpeedLowSpeedBrakeTest.ToolScalingDivisor :=1;
bogLimitSpeedLowSpeedBrakeTest.ToolScalingMultiplier :=1;
bogLimitSpeedLowSpeedBrakeTest.ToolScalingOffset :=0;
bogLimitSpeedLowSpeedBrakeTest.ToolUnit :="";

bogSlopeSensorFault.AppScalingDivisor :=1;
bogSlopeSensorFault.AppScalingMultiplier :=1;
bogSlopeSensorFault.AppScalingOffset :=0;
bogSlopeSensorFault.AppUnit :="";
bogSlopeSensorFault.CanDefault :=0;
bogSlopeSensorFault.CanInit :=0;
bogSlopeSensorFault.CanMax :=1;
bogSlopeSensorFault.CanMin :=0;
bogSlopeSensorFault.CanUnit :="";
bogSlopeSensorFault.Description :="Fuel low";
bogSlopeSensorFault.ErrorReaction := eErrorReaction.ERSIG_DFLT;
bogSlopeSensorFault.ReceiverAdress :=1;
bogSlopeSensorFault.ToolScalingDivisor :=1;
bogSlopeSensorFault.ToolScalingMultiplier :=1;
bogSlopeSensorFault.ToolScalingOffset :=0;
bogSlopeSensorFault.ToolUnit :="";

bogMastMeasureFault.AppScalingDivisor :=1;
bogMastMeasureFault.AppScalingMultiplier :=1;
bogMastMeasureFault.AppScalingOffset :=0;
bogMastMeasureFault.AppUnit :="";
bogMastMeasureFault.CanDefault :=0;
bogMastMeasureFault.CanInit :=0;
bogMastMeasureFault.CanMax :=1;
bogMastMeasureFault.CanMin :=0;
bogMastMeasureFault.CanUnit :="";
bogMastMeasureFault.Description :="Mast Measure Fault";
bogMastMeasureFault.ErrorReaction := eErrorReaction.ERSIG_DFLT;
bogMastMeasureFault.ReceiverAdress :=1;
bogMastMeasureFault.ToolScalingDivisor :=1;
bogMastMeasureFault.ToolScalingMultiplier :=1;
bogMastMeasureFault.ToolScalingOffset :=0;
bogMastMeasureFault.ToolUnit :="";

i16gEncodeurTurretAngle.AppScalingDivisor :=1;
i16gEncodeurTurretAngle.AppScalingMultiplier :=1;
i16gEncodeurTurretAngle.AppScalingOffset :=0;
i16gEncodeurTurretAngle.AppUnit :="";
i16gEncodeurTurretAngle.CanDefault :=0;
i16gEncodeurTurretAngle.CanInit :=0;
i16gEncodeurTurretAngle.CanMax :=VBasic.LibConst.I16_MAX;
i16gEncodeurTurretAngle.CanMin :=VBasic.LibConst.I16_MIN;
i16gEncodeurTurretAngle.CanUnit :="";
i16gEncodeurTurretAngle.Description :="RPM Solenoid value";
i16gEncodeurTurretAngle.ErrorReaction := eErrorReaction.ERSIG_DFLT;
i16gEncodeurTurretAngle.ReceiverAdress :=1;
i16gEncodeurTurretAngle.ToolScalingDivisor :=1;
i16gEncodeurTurretAngle.ToolScalingMultiplier :=1;
i16gEncodeurTurretAngle.ToolScalingOffset :=0;
i16gEncodeurTurretAngle.ToolUnit :="";


                
END_METHOD
END_FUNCTION_BLOCK

FUNCTION_BLOCK Msg2C0SendToEvision7MessageClass EXTENDS CanReceiveMessageClass
  VAR_INPUT
    u16gEngine_Use_Time : UInt16CanSignalClass;
    u16gEngine_RPM : UInt16CanSignalClass;
    u16gVehiculeSpeed : UInt16CanSignalClass;
    u8gLateralizationStop : UInt8CanSignalClass;
    u8gKeySelector : UInt8CanSignalClass;
    Counter : UInt32CanSignalClass;
  END_VAR

            
          

METHOD SetData
  VAR_INPUT
    CanMsgPointer : POINTER TO CanMessageClass;
  END_VAR
                  IF IsValidPointer(canMsgPointer,'SetData') THEN
	SUPER^.SetData(CanMsgPointer);
	//Set the new data
	u16gEngine_Use_Time.Value := canMsgPointer^.GetUint16(0);
	u16gEngine_RPM.Value := canMsgPointer^.GetUint16(16);
	u16gVehiculeSpeed.Value := canMsgPointer^.GetUint16(32);
	u8gLateralizationStop.Value := canMsgPointer^.GetUint8(48);
	u8gKeySelector.Value := canMsgPointer^.GetUint8(56);
	//And increase the counter
	Counter.Value := CanMsgPointer^.Counter.Value;
END_IF

                
END_METHOD

PROPERTY u16gEngine_Use_TimeRawValue : UINT
GET
                    IF u16gEngine_Use_Time.AppScalingMultiplier = 0 THEN
	_MatchLog^.Error("Get u16gEngine_Use_TimeRawValue", "Division by Zero!");
	RETURN;
End_IF

u16gEngine_Use_TimeRawValue := TO_UINT((u16gEngine_Use_Time.Value - u16gEngine_Use_Time.AppScalingOffset) * u16gEngine_Use_Time.AppScalingDivisor / u16gEngine_Use_Time.AppScalingMultiplier);

                  
END_GET
END_PROPERTY

PROPERTY u16gEngine_RPMRawValue : UINT
GET
                    IF u16gEngine_RPM.AppScalingMultiplier = 0 THEN
	_MatchLog^.Error("Get u16gEngine_RPMRawValue", "Division by Zero!");
	RETURN;
End_IF

u16gEngine_RPMRawValue := TO_UINT((u16gEngine_RPM.Value - u16gEngine_RPM.AppScalingOffset) * u16gEngine_RPM.AppScalingDivisor / u16gEngine_RPM.AppScalingMultiplier);

                  
END_GET
END_PROPERTY

PROPERTY u16gVehiculeSpeedRawValue : UINT
GET
                    IF u16gVehiculeSpeed.AppScalingMultiplier = 0 THEN
	_MatchLog^.Error("Get u16gVehiculeSpeedRawValue", "Division by Zero!");
	RETURN;
End_IF

u16gVehiculeSpeedRawValue := TO_UINT((u16gVehiculeSpeed.Value - u16gVehiculeSpeed.AppScalingOffset) * u16gVehiculeSpeed.AppScalingDivisor / u16gVehiculeSpeed.AppScalingMultiplier);

                  
END_GET
END_PROPERTY

PROPERTY u8gLateralizationStopRawValue : USINT
GET
                    IF u8gLateralizationStop.AppScalingMultiplier = 0 THEN
	_MatchLog^.Error("Get u8gLateralizationStopRawValue", "Division by Zero!");
	RETURN;
End_IF

u8gLateralizationStopRawValue := TO_USINT((u8gLateralizationStop.Value - u8gLateralizationStop.AppScalingOffset) * u8gLateralizationStop.AppScalingDivisor / u8gLateralizationStop.AppScalingMultiplier);

                  
END_GET
END_PROPERTY

PROPERTY u8gKeySelectorRawValue : USINT
GET
                    IF u8gKeySelector.AppScalingMultiplier = 0 THEN
	_MatchLog^.Error("Get u8gKeySelectorRawValue", "Division by Zero!");
	RETURN;
End_IF

u8gKeySelectorRawValue := TO_USINT((u8gKeySelector.Value - u8gKeySelector.AppScalingOffset) * u8gKeySelector.AppScalingDivisor / u8gKeySelector.AppScalingMultiplier);

                  
END_GET
END_PROPERTY

PROPERTY u16gEngine_Use_TimeToolValue : UINT
GET
                    IF u16gEngine_Use_Time.ToolScalingDivisor = 0 OR u16gEngine_Use_Time.AppScalingMultiplier = 0 THEN
	_MatchLog^.Error("Get u16gEngine_Use_TimeToolValue", "Division by Zero!");
	RETURN;
END_IF

u16gEngine_Use_TimeToolValue := TO_UINT(((u16gEngine_Use_Time.Value - u16gEngine_Use_Time.AppScalingOffset) * u16gEngine_Use_Time.AppScalingDivisor / u16gEngine_Use_Time.AppScalingMultiplier * u16gEngine_Use_Time.ToolScalingMultiplier / u16gEngine_Use_Time.ToolScalingDivisor) + u16gEngine_Use_Time.ToolScalingOffset);

                  
END_GET
END_PROPERTY

PROPERTY u16gEngine_RPMToolValue : UINT
GET
                    IF u16gEngine_RPM.ToolScalingDivisor = 0 OR u16gEngine_RPM.AppScalingMultiplier = 0 THEN
	_MatchLog^.Error("Get u16gEngine_RPMToolValue", "Division by Zero!");
	RETURN;
END_IF

u16gEngine_RPMToolValue := TO_UINT(((u16gEngine_RPM.Value - u16gEngine_RPM.AppScalingOffset) * u16gEngine_RPM.AppScalingDivisor / u16gEngine_RPM.AppScalingMultiplier * u16gEngine_RPM.ToolScalingMultiplier / u16gEngine_RPM.ToolScalingDivisor) + u16gEngine_RPM.ToolScalingOffset);

                  
END_GET
END_PROPERTY

PROPERTY u16gVehiculeSpeedToolValue : UINT
GET
                    IF u16gVehiculeSpeed.ToolScalingDivisor = 0 OR u16gVehiculeSpeed.AppScalingMultiplier = 0 THEN
	_MatchLog^.Error("Get u16gVehiculeSpeedToolValue", "Division by Zero!");
	RETURN;
END_IF

u16gVehiculeSpeedToolValue := TO_UINT(((u16gVehiculeSpeed.Value - u16gVehiculeSpeed.AppScalingOffset) * u16gVehiculeSpeed.AppScalingDivisor / u16gVehiculeSpeed.AppScalingMultiplier * u16gVehiculeSpeed.ToolScalingMultiplier / u16gVehiculeSpeed.ToolScalingDivisor) + u16gVehiculeSpeed.ToolScalingOffset);

                  
END_GET
END_PROPERTY

PROPERTY u8gLateralizationStopToolValue : USINT
GET
                    IF u8gLateralizationStop.ToolScalingDivisor = 0 OR u8gLateralizationStop.AppScalingMultiplier = 0 THEN
	_MatchLog^.Error("Get u8gLateralizationStopToolValue", "Division by Zero!");
	RETURN;
END_IF

u8gLateralizationStopToolValue := TO_USINT(((u8gLateralizationStop.Value - u8gLateralizationStop.AppScalingOffset) * u8gLateralizationStop.AppScalingDivisor / u8gLateralizationStop.AppScalingMultiplier * u8gLateralizationStop.ToolScalingMultiplier / u8gLateralizationStop.ToolScalingDivisor) + u8gLateralizationStop.ToolScalingOffset);

                  
END_GET
END_PROPERTY

PROPERTY u8gKeySelectorToolValue : USINT
GET
                    IF u8gKeySelector.ToolScalingDivisor = 0 OR u8gKeySelector.AppScalingMultiplier = 0 THEN
	_MatchLog^.Error("Get u8gKeySelectorToolValue", "Division by Zero!");
	RETURN;
END_IF

u8gKeySelectorToolValue := TO_USINT(((u8gKeySelector.Value - u8gKeySelector.AppScalingOffset) * u8gKeySelector.AppScalingDivisor / u8gKeySelector.AppScalingMultiplier * u8gKeySelector.ToolScalingMultiplier / u8gKeySelector.ToolScalingDivisor) + u8gKeySelector.ToolScalingOffset);

                  
END_GET
END_PROPERTY

METHOD InitializeCanSignals
                  u16gEngine_Use_Time.AppScalingDivisor :=1;
u16gEngine_Use_Time.AppScalingMultiplier :=1;
u16gEngine_Use_Time.AppScalingOffset :=0;
u16gEngine_Use_Time.AppUnit :="";
u16gEngine_Use_Time.CanDefault :=0;
u16gEngine_Use_Time.CanInit :=0;
u16gEngine_Use_Time.CanMax :=VBasic.LibConst.U16_MAX;
u16gEngine_Use_Time.CanMin :=VBasic.LibConst.U16_MIN;
u16gEngine_Use_Time.CanUnit :="";
u16gEngine_Use_Time.Description :="Engine use time in hour";
u16gEngine_Use_Time.ErrorReaction := eErrorReaction.ERSIG_DFLT;
u16gEngine_Use_Time.ReceiverAdress :=1;
u16gEngine_Use_Time.ToolScalingDivisor :=1;
u16gEngine_Use_Time.ToolScalingMultiplier :=1;
u16gEngine_Use_Time.ToolScalingOffset :=0;
u16gEngine_Use_Time.ToolUnit :="";

u16gEngine_RPM.AppScalingDivisor :=1;
u16gEngine_RPM.AppScalingMultiplier :=1;
u16gEngine_RPM.AppScalingOffset :=0;
u16gEngine_RPM.AppUnit :="";
u16gEngine_RPM.CanDefault :=0;
u16gEngine_RPM.CanInit :=0;
u16gEngine_RPM.CanMax :=VBasic.LibConst.U16_MAX;
u16gEngine_RPM.CanMin :=VBasic.LibConst.U16_MIN;
u16gEngine_RPM.CanUnit :="";
u16gEngine_RPM.Description :="Engine RPM";
u16gEngine_RPM.ErrorReaction := eErrorReaction.ERSIG_DFLT;
u16gEngine_RPM.ReceiverAdress :=1;
u16gEngine_RPM.ToolScalingDivisor :=1;
u16gEngine_RPM.ToolScalingMultiplier :=1;
u16gEngine_RPM.ToolScalingOffset :=0;
u16gEngine_RPM.ToolUnit :="";

u16gVehiculeSpeed.AppScalingDivisor :=1;
u16gVehiculeSpeed.AppScalingMultiplier :=1;
u16gVehiculeSpeed.AppScalingOffset :=0;
u16gVehiculeSpeed.AppUnit :="";
u16gVehiculeSpeed.CanDefault :=0;
u16gVehiculeSpeed.CanInit :=0;
u16gVehiculeSpeed.CanMax :=VBasic.LibConst.U16_MAX;
u16gVehiculeSpeed.CanMin :=VBasic.LibConst.U16_MIN;
u16gVehiculeSpeed.CanUnit :="";
u16gVehiculeSpeed.Description :="Vehicule Speed in Km/h * 100";
u16gVehiculeSpeed.ErrorReaction := eErrorReaction.ERSIG_DFLT;
u16gVehiculeSpeed.ReceiverAdress :=1;
u16gVehiculeSpeed.ToolScalingDivisor :=1;
u16gVehiculeSpeed.ToolScalingMultiplier :=1;
u16gVehiculeSpeed.ToolScalingOffset :=0;
u16gVehiculeSpeed.ToolUnit :="";

u8gLateralizationStop.AppScalingDivisor :=1;
u8gLateralizationStop.AppScalingMultiplier :=1;
u8gLateralizationStop.AppScalingOffset :=0;
u8gLateralizationStop.AppUnit :="";
u8gLateralizationStop.CanDefault :=0;
u8gLateralizationStop.CanInit :=0;
u8gLateralizationStop.CanMax :=VBasic.LibConst.U8_MAX;
u8gLateralizationStop.CanMin :=VBasic.LibConst.U8_MIN;
u8gLateralizationStop.CanUnit :="";
u8gLateralizationStop.Description :="Lateralization Stop 1=bi lateralization 2=ALO Work 3=Multiple track (A3)";
u8gLateralizationStop.ErrorReaction := eErrorReaction.ERSIG_DFLT;
u8gLateralizationStop.ReceiverAdress :=1;
u8gLateralizationStop.ToolScalingDivisor :=1;
u8gLateralizationStop.ToolScalingMultiplier :=1;
u8gLateralizationStop.ToolScalingOffset :=0;
u8gLateralizationStop.ToolUnit :="";

u8gKeySelector.AppScalingDivisor :=1;
u8gKeySelector.AppScalingMultiplier :=1;
u8gKeySelector.AppScalingOffset :=0;
u8gKeySelector.AppUnit :="";
u8gKeySelector.CanDefault :=0;
u8gKeySelector.CanInit :=0;
u8gKeySelector.CanMax :=VBasic.LibConst.U8_MAX;
u8gKeySelector.CanMin :=VBasic.LibConst.U8_MIN;
u8gKeySelector.CanUnit :="";
u8gKeySelector.Description :="Key Selector 1=bi lateralization 2=ALO Work 3=Multiple track(A6)";
u8gKeySelector.ErrorReaction := eErrorReaction.ERSIG_DFLT;
u8gKeySelector.ReceiverAdress :=1;
u8gKeySelector.ToolScalingDivisor :=1;
u8gKeySelector.ToolScalingMultiplier :=1;
u8gKeySelector.ToolScalingOffset :=0;
u8gKeySelector.ToolUnit :="";


                
END_METHOD
END_FUNCTION_BLOCK

FUNCTION_BLOCK Msg3C0SendToEvision7MessageClass EXTENDS CanReceiveMessageClass
  VAR_INPUT
    u16gFrontSpeedRailWayAxle : UInt16CanSignalClass;
    u16gBackSpeedRailWayAxle : UInt16CanSignalClass;
    u16gAvdvancePeriod : UInt16CanSignalClass;
    u16gPressureEfficiencyRate : UInt16CanSignalClass;
    Counter : UInt32CanSignalClass;
  END_VAR

            
          

METHOD SetData
  VAR_INPUT
    CanMsgPointer : POINTER TO CanMessageClass;
  END_VAR
                  IF IsValidPointer(canMsgPointer,'SetData') THEN
	SUPER^.SetData(CanMsgPointer);
	//Set the new data
	u16gFrontSpeedRailWayAxle.Value := canMsgPointer^.GetUint16(0);
	u16gBackSpeedRailWayAxle.Value := canMsgPointer^.GetUint16(16);
	u16gAvdvancePeriod.Value := canMsgPointer^.GetUint16(32);
	u16gPressureEfficiencyRate.Value := canMsgPointer^.GetUint16(48);
	//And increase the counter
	Counter.Value := CanMsgPointer^.Counter.Value;
END_IF

                
END_METHOD

PROPERTY u16gFrontSpeedRailWayAxleRawValue : UINT
GET
                    IF u16gFrontSpeedRailWayAxle.AppScalingMultiplier = 0 THEN
	_MatchLog^.Error("Get u16gFrontSpeedRailWayAxleRawValue", "Division by Zero!");
	RETURN;
End_IF

u16gFrontSpeedRailWayAxleRawValue := TO_UINT((u16gFrontSpeedRailWayAxle.Value - u16gFrontSpeedRailWayAxle.AppScalingOffset) * u16gFrontSpeedRailWayAxle.AppScalingDivisor / u16gFrontSpeedRailWayAxle.AppScalingMultiplier);

                  
END_GET
END_PROPERTY

PROPERTY u16gBackSpeedRailWayAxleRawValue : UINT
GET
                    IF u16gBackSpeedRailWayAxle.AppScalingMultiplier = 0 THEN
	_MatchLog^.Error("Get u16gBackSpeedRailWayAxleRawValue", "Division by Zero!");
	RETURN;
End_IF

u16gBackSpeedRailWayAxleRawValue := TO_UINT((u16gBackSpeedRailWayAxle.Value - u16gBackSpeedRailWayAxle.AppScalingOffset) * u16gBackSpeedRailWayAxle.AppScalingDivisor / u16gBackSpeedRailWayAxle.AppScalingMultiplier);

                  
END_GET
END_PROPERTY

PROPERTY u16gAvdvancePeriodRawValue : UINT
GET
                    IF u16gAvdvancePeriod.AppScalingMultiplier = 0 THEN
	_MatchLog^.Error("Get u16gAvdvancePeriodRawValue", "Division by Zero!");
	RETURN;
End_IF

u16gAvdvancePeriodRawValue := TO_UINT((u16gAvdvancePeriod.Value - u16gAvdvancePeriod.AppScalingOffset) * u16gAvdvancePeriod.AppScalingDivisor / u16gAvdvancePeriod.AppScalingMultiplier);

                  
END_GET
END_PROPERTY

PROPERTY u16gPressureEfficiencyRateRawValue : UINT
GET
                    IF u16gPressureEfficiencyRate.AppScalingMultiplier = 0 THEN
	_MatchLog^.Error("Get u16gPressureEfficiencyRateRawValue", "Division by Zero!");
	RETURN;
End_IF

u16gPressureEfficiencyRateRawValue := TO_UINT((u16gPressureEfficiencyRate.Value - u16gPressureEfficiencyRate.AppScalingOffset) * u16gPressureEfficiencyRate.AppScalingDivisor / u16gPressureEfficiencyRate.AppScalingMultiplier);

                  
END_GET
END_PROPERTY

PROPERTY u16gFrontSpeedRailWayAxleToolValue : UINT
GET
                    IF u16gFrontSpeedRailWayAxle.ToolScalingDivisor = 0 OR u16gFrontSpeedRailWayAxle.AppScalingMultiplier = 0 THEN
	_MatchLog^.Error("Get u16gFrontSpeedRailWayAxleToolValue", "Division by Zero!");
	RETURN;
END_IF

u16gFrontSpeedRailWayAxleToolValue := TO_UINT(((u16gFrontSpeedRailWayAxle.Value - u16gFrontSpeedRailWayAxle.AppScalingOffset) * u16gFrontSpeedRailWayAxle.AppScalingDivisor / u16gFrontSpeedRailWayAxle.AppScalingMultiplier * u16gFrontSpeedRailWayAxle.ToolScalingMultiplier / u16gFrontSpeedRailWayAxle.ToolScalingDivisor) + u16gFrontSpeedRailWayAxle.ToolScalingOffset);

                  
END_GET
END_PROPERTY

PROPERTY u16gBackSpeedRailWayAxleToolValue : UINT
GET
                    IF u16gBackSpeedRailWayAxle.ToolScalingDivisor = 0 OR u16gBackSpeedRailWayAxle.AppScalingMultiplier = 0 THEN
	_MatchLog^.Error("Get u16gBackSpeedRailWayAxleToolValue", "Division by Zero!");
	RETURN;
END_IF

